# B&R Automation Studio project NewPendant_NG4_11_05_25A (part 7)

```c
				// Dodane - Nie ma Xcmd Stop w TRVL_BPV_POS
				if((TVL_ROT_Param_Set[0].Mode == 2) // with only position
					|| (TVL_ROT_Param_Set[0].Mode == 3)) // with interrupt
					Process[m->pCfg->HeadCfg.TVL.PROC_Indx].xCMD = 0;
			}
			*/

///////////////////////////////////////////////////////////////////////////
/// Nowosc Index wczesniej

			if((curCalib->GenSetup[SETUP_EXTRAS]&0x4)){

				switch(curCalib->GenSetup[SETUP_HEAD_SETUP] ){

						default:

							if(curCalib->GenSetup[SETUP_INDX_ENBL] == 3){ // In OSc

								if(INDEX_Param_Set[0].pStepDist){

									Process[m->pCfg->HeadCfg.OSC.PROC_Indx].xCMD = prcsSTEPneg; // Quick Step with delay

									if(curCalib->GenSetup[SETUP_INDX_DIR])
										Process[m->pCfg->HeadCfg.OSC.PROC_Indx].fParam[1] = (*INDEX_Param_Set[0].pStepDist);
									else
										Process[m->pCfg->HeadCfg.OSC.PROC_Indx].fParam[1] = (*INDEX_Param_Set[0].pStepDist) * (-1.0);

									KK_Catched = 133;

									//m->SeqStep++;
								}
								//else
									//m->SeqStep = 203;

							}

							else if(curCalib->GenSetup[SETUP_INDX_ENBL] == 1){

								if(INDEX_Param_Set[0].pStepDist){
									Process[m->pCfg->HeadCfg.INDX.PROC_Indx].xCMD = prcsSTEPpos;

									if(curCalib->GenSetup[SETUP_INDX_DIR])
										Process[m->pCfg->HeadCfg.INDX.PROC_Indx].fParam[1] = (*INDEX_Param_Set[0].pStepDist);
									else
										Process[m->pCfg->HeadCfg.INDX.PROC_Indx].fParam[1] = (*INDEX_Param_Set[0].pStepDist) * (-1.0);

									m->SeqStep++;

								}
								//else
									//m->SeqStep = 203;

							}
							//else
								//m->SeqStep = 203;

						break;

					}

			}

/////////////////////////////////////////////////////////////////////////
#ifdef EXTENDED_LOGS

			LogTxt(&LogMgr, "Path %d Done: %.2f" , (UDINT)File_RW._int.PathDoneCnt, ABS_TVL_Pos);
#else
			LogTxt(&LogMgr, "Path %d Done" , (UDINT)File_RW._int.PathDoneCnt);

#endif

			//TimerStart(&WF_Catch_TMR, curCfg->Param[parWF_RampDwn].val[0]);
			m->SeqStep++;

		break;

		case 201:

			// Always Coolant On
			if (!m->TestMode)
			{
				if (Process[m->pCfg->HeadCfg.COOL.PROC_Indx].Status != prcsSTATUS_Run)
					Process[m->pCfg->HeadCfg.COOL.PROC_Indx].xCMD = prcsSTART;
			}

			ret = 5; // Preparing To Stop

			if (StopBtn)
			{
#ifdef EXTENDED_LOGS

				LogTxt(&LogMgr, "Quick stop %.2f" , ABS_TVL_Pos);
#else
				LogTxt(&LogMgr, "Quick stop");
#endif
				m->SeqStep = 254;			// Quick Stop
			}

			status = 1;

			if (Process[m->pCfg->HeadCfg.TVL.PROC_Indx].Status != prcsSTATUS_Stopped){ // stopped by end of travel
				status = 0;
			}
			if (Process[m->pCfg->HeadCfg.OSC.PROC_Indx].Status != prcsSTATUS_Stopped)
				status = 0;

			if (Process[m->pCfg->HeadCfg.AVC.PROC_Indx].Status != prcsSTATUS_Stopped)
				status = 0;

			if (Process[m->pCfg->HeadCfg.WF.PROC_Indx].Status != prcsSTATUS_Stopped)
				status = 0;

			//if (Process[m->pCfg->HeadCfg.GAS.PROC_Indx].Status != prcsSTATUS_Stopped)
				//status = 0;

			if (Process[m->pCfg->HeadCfg.WP.PROC_Indx].Status != prcsSTATUS_Stopped)
				status = 0;

			if (Process[m->pCfg->HeadCfg.TIG.PROC_Indx].Status != prcsSTATUS_Stopped)
				status = 0;

			if (Process[m->pCfg->HeadCfg.HW.PROC_Indx].Status != prcsSTATUS_Stopped)
				status = 0;

			if (status)
			{

#ifdef EXTENDED_LOGS

				LogTxt(&LogMgr, "M:All%d Stop: %.2f" ,(UDINT) m->ToolHeadID, ABS_TVL_Pos);

#endif

				if(!(curCalib->GenSetup[SETUP_EXTRAS]&0x4)){

					switch(curCalib->GenSetup[SETUP_HEAD_SETUP] ){

						/*
						case BPV_v2_MPGH:
						case BPV_v2_MPGV:

						case BPV_v2_MPBO:

							if(curCalib->GenSetup[SETUP_INDX_ENBL] == 3){ // In OSc

								if(INDEX_Param_Set[0].pStepDist){

									Process[m->pCfg->HeadCfg.OSC.PROC_Indx].xCMD = prcsSTEPpos;

									if(curCalib->GenSetup[SETUP_INDX_DIR])
										Process[m->pCfg->HeadCfg.OSC.PROC_Indx].fParam[1] = (*INDEX_Param_Set[0].pStepDist);
									else
										Process[m->pCfg->HeadCfg.OSC.PROC_Indx].fParam[1] = (*INDEX_Param_Set[0].pStepDist) * (-1.0);

									KK_Catched = 133;

									m->SeqStep++;
								}
								else
									m->SeqStep = 203;

							}
							else
								m->SeqStep = 203;

						break;
						*/

						default:

							if(curCalib->GenSetup[SETUP_INDX_ENBL] == 3){ // In OSc

								if(INDEX_Param_Set[0].pStepDist){

									Process[m->pCfg->HeadCfg.OSC.PROC_Indx].xCMD = prcsSTEPpos;

									if(curCalib->GenSetup[SETUP_INDX_DIR])
										Process[m->pCfg->HeadCfg.OSC.PROC_Indx].fParam[1] = (*INDEX_Param_Set[0].pStepDist);
									else
										Process[m->pCfg->HeadCfg.OSC.PROC_Indx].fParam[1] = (*INDEX_Param_Set[0].pStepDist) * (-1.0);

									KK_Catched = 133;

									m->SeqStep++;
								}
								else
									m->SeqStep = 203;

							}

							else if(curCalib->GenSetup[SETUP_INDX_ENBL] == 1){

								if(INDEX_Param_Set[0].pStepDist){
									Process[m->pCfg->HeadCfg.INDX.PROC_Indx].xCMD = prcsSTEPpos;

									if(curCalib->GenSetup[SETUP_INDX_DIR])
										Process[m->pCfg->HeadCfg.INDX.PROC_Indx].fParam[1] = (*INDEX_Param_Set[0].pStepDist);
									else
										Process[m->pCfg->HeadCfg.INDX.PROC_Indx].fParam[1] = (*INDEX_Param_Set[0].pStepDist) * (-1.0);

									m->SeqStep++;

								}
								else
									m->SeqStep = 203;

							}
							else
								m->SeqStep = 203;

						break;

					}

					}

			}

		break;

		case 202:

			// Always Coolant On
			if (!m->TestMode)
			{
				if (Process[m->pCfg->HeadCfg.COOL.PROC_Indx].Status != prcsSTATUS_Run)
					Process[m->pCfg->HeadCfg.COOL.PROC_Indx].xCMD = prcsSTART;
			}

			if (StopBtn)
			{
				LogTxt(&LogMgr, "Quick stop");

				m->SeqStep			= 254;			// Quick Stop
				break;
			}

			if(Process[m->pCfg->HeadCfg.INDX.PROC_Indx].Status == prcsSTATUS_Stopped
				&& Process[m->pCfg->HeadCfg.OSC.PROC_Indx].Status == prcsSTATUS_Stopped){

				TimerStart(&m->sm.Tmr1, 0.1);
				m->SeqStep++;

			}

		break;

		case 203:
			// Always Coolant On
			if (StopBtn)
			{
				LogTxt(&LogMgr, "Halt stop");

				m->SeqStep			= 254;			// Quick Stop
				break;
			}

			if (!m->TestMode)
			{
				if (Process[m->pCfg->HeadCfg.COOL.PROC_Indx].Status != prcsSTATUS_Run)
					Process[m->pCfg->HeadCfg.COOL.PROC_Indx].xCMD = prcsSTART;
			}

			if(Process[m->pCfg->HeadCfg.TVL.PROC_Indx].Status == prcsSTATUS_Stopped){

				LogTxt(&LogMgr, "M: Cyc. Time %.2f" , GlobalTimer);
				m->SeqStep++;
			}

		break;

		case 204:

			// Always Coolant On
			if (!m->TestMode)
			{
				if (Process[m->pCfg->HeadCfg.COOL.PROC_Indx].Status != prcsSTATUS_Run)
					Process[m->pCfg->HeadCfg.COOL.PROC_Indx].xCMD = prcsSTART;
			}

			ret = 5; // Preparing To Stop

			if (StopBtn)
			{
				LogTxt(&LogMgr, "Quick stop");
				m->SeqStep = 254;			// Quick Stop
				//m->SeqStep = 205;			// Normal Stop
				break;
			}

			// Check if Index move done
			if (1)
			{

				if((abs(m->curSegm[ACT_TVL_DIST] - Process[m->pCfg->HeadCfg.TVL.PROC_Indx].Param[3]) < 10)
				//if((Process[m->pCfg->HeadCfg.TVL.PROC_Indx].Status == prcsSTATUS_Stopped)
					&& (m->SubSeqStep == 2)) // IMPORTANT - head swap is only when was rewrap before
				{

					m->SubSeqStep = 1;

					if (curCfg->Param_ENUM[parENUM_PathMode].val[0] == 0.0)
						m->ToolHeadID = !m->ToolHeadID;

					if (curCfg->Param_ENUM[parENUM_TVL_MODE].val[0] == 0)
					{ // Relative Move
						if (TVL_ROT_Param_Set[0].pEncoder)
							OLD_MTR_POS[TVL_ENC_HOME] = *TVL_ROT_Param_Set[0].pEncoder;
					}
					AutoStartEnable = 1;
					m->SeqStep++;

				}

				else
				{
					m->SeqStep = 254;
				}

			}

		break;

		case 205:

			if(curCfg->Param[parGEN_WeldProgramRepeat].val[0] > 0)
				File_RW._int.PathDoneCnt++;
			else
				File_RW._int.PathDoneCnt = 0;

			newFile = 0;

			if (curCfg->Param_ENUM[parENUM_WeldProgramLinkMode].val[0] > 0.0)
			{

				if (curCfg->Param[parGEN_WeldProgramRepeat].val[0] == 0.0)
				{

					if (strlen(curCfg->NextProgramName) > 0)
					{

						if (!strstr(curCfg->NextProgramName, "NONE"))
						{ // Not None
							TakeNextWeldProgram(hmi);
							newFile 			= 1;

						}

					}

				}

				else
				{

					if (File_RW._int.PathDoneCnt > (UINT)curCfg->Param[parGEN_WeldProgramRepeat].val[0] )
					{

						if (strlen(curCfg->NextProgramName) > 0)
						{

							if (!strstr(curCfg->NextProgramName, "NONE"))
							{ // Not None
								TakeNextWeldProgram(hmi);
								newFile 			= 1;
							}

						}

					}

				}

			}

			if (newFile)
				m->SeqStep = 206;
			else
				m->SeqStep = 207;

		break;

		case 206:
			if (File_RW.CMD == 0)
			{

				if (File_RW.Error)
					m->SeqStep = 206;

				else
				{
					AutoStartEnable = 1;
					m->SeqStep = 207;

				}
			}

		break;

		case 207:

			AutoStartEnable = 1;

			if (File_RW._int.PathDoneCnt > (UINT)curCfg->Param[parGEN_WeldProgramRepeat].val[0] )
			{
				File_RW._int.PathDoneCnt = (UINT)curCfg->Param[parGEN_WeldProgramRepeat].val[0];

				AutoStartEnable 	= 0;
			}

			m->SeqStep++;

		break;

		case 208:
			///////////////////////////////////
			//Auto Start
			if (curCalib->GenSetup[SETUP_AUTO_START] && AutoStartEnable)
			{
				TimerStart(&m->sm.Tmr1, curCalib->GenFloatValue[SETUP_FLOAT_AUTOSTART_DLY]);
				m->SeqStep = 220;

			}
			else
				m->SeqStep = 254;

		break;

		case 210:

			if (StopBtn)
			{
				LogTxt(&LogMgr, "Quick stop");

				m->SeqStep = 254;			// Quick Stop

			}
			else if (Process[m->pCfg->HeadCfg.TVL.PROC_Indx].Status == prcsSTATUS_Stopped) // stopped by end of travel
				m->SeqStep = 0;

		break;

		case 220:

			if (StopBtn)
			{
				LogTxt(&LogMgr, "Quick stop");

				m->SeqStep = 254;			// Quick Stop
				break;
			}
			else if(!TimerIsTimeOut(&m->sm.Tmr1))
				break;

			GlobalTimer = 0;

			//WF_TVL_Diff = 0;
			LogTxt(&LogMgr, "Auto Repeat");
			AutoStartBtn = 1;
			m->SeqStep = 0;

		break;

		case 254:

			for (i = 0; i < PROCESS_NUM; i++)
			{ // beside PROC_COOL
				if (i != PROC_COOL)
					Process[i].xCMD = prcsHalt;
			}

			Process[m->pCfg->HeadCfg.OSC.PROC_Indx].Param[0] = 1; // STop without ramp
			Process[m->pCfg->HeadCfg.OSC.PROC_Indx].xCMD = prcsQuickSTOP; // return to center position
			Process[m->pCfg->HeadCfg.GAS.PROC_Indx].xCMD = prcsSTOP; // maintain gas
			m->SeqStep++;

		break;

		default:

			if(curCfg->Param_ENUM[parENUM_AVC_Mode].val[0] != 3) // AVC Mode NOT LOCKED !
				Process[m->pCfg->HeadCfg.AVC.PROC_Indx].Param[0] = 0;

			if (StopBtn)
			{
				LogTxt(&LogMgr, "Halt stop");

				for (i = 0; i < PROCESS_NUM; i++)
				{ // beside PROC_COOL
					if (i!= PROC_COOL && i!= PROC_OSC)
						Process[i].xCMD = prcsHalt;
				}

				Process[m->pCfg->HeadCfg.GAS.PROC_Indx].xCMD = prcsSTOP; // maintain gas
				m->SeqStep			= 0;

			}

			if (Process[m->pCfg->HeadCfg.OSC.PROC_Indx].Status == prcsSTATUS_Stopped)
				m->SeqStep = 0;

			if (m->SeqStep == 0)
			{
				// Load new AVC param from new file
				TML_MTR_INST[m->pCfg->HeadCfg.AVC.TML_A_Indx]._cfg.signFilter =	curCfg->Param[parAVC_FbkFilter].val[0];
			}

		break;

		}

		//if((Process[m->pCfg->HeadCfg.TVL.PROC_Indx].Status == prcsSTATUS_Stopped))
		//StopBtn_Latch = 0;
		////////////////////////////
		TimerExecute(&WireDisable_TMR);
		TimerExecute(&WF_Catch_TMR);

		return ret;
	}

		/*********************************************************/
			/****	Process parameters assigments	************************/

	DINT MasterSequence_Contin_OneWay_dobra_alebezWeldIndex(MASTER_typ * m, HMI_typ * hmi, plcbit StartBtn, plcbit StopBtn)
	{
	int 			i;
	char			status;
	DINT			ret;
	DINT			d;
	USINT			newFile;

	//Cfg_typ *cfg;
	CurCfg_typ *	curCfg;

	//CurCalib_typ *curCalib , *defCalib;
	//Scaled_Var_obj *var;
	//cfg = (Cfg_typ*) m->pCfg;
	curCfg				= (CurCfg_typ *)
	m->pCurCfg;

	//curCalib = (CurCalib_typ*) m->pCalib;
	//defCalib = (CurCalib_typ*) m->pDefaultCalib;
	//var = (Scaled_Var_obj*) m->pScaledVar;
	m->TestMode 		= intrf->TestMode;

	ret 				= 0;

	if((hmi->curHeadID == 0xFFFE)){ // Screen RUn or Alter Run

		if(intrf->GlblBtnCmd[0] &ANDR_BTN_UP){

			AVC_Param_Set[0].BoostCmd = 1;
			PS_Param_Set[0].BoostCmd = 1;
			TVL_ROT_Param_Set[0].BoostCmd = 1;
			WIRE_Param_Set[0].BoostCmd = 1;
			WIRE_Param_Set[1].BoostCmd = 1;

		}
		else if(intrf->GlblBtnCmd[0] &ANDR_BTN_DOWN){

			AVC_Param_Set[0].BoostCmd = 2;
			PS_Param_Set[0].BoostCmd = 2;
			TVL_ROT_Param_Set[0].BoostCmd = 2;
			WIRE_Param_Set[0].BoostCmd = 2;
			WIRE_Param_Set[1].BoostCmd = 2;

		}
		else{

			AVC_Param_Set[0].BoostCmd = 0;
			PS_Param_Set[0].BoostCmd = 0;
			TVL_ROT_Param_Set[0].BoostCmd = 0;
			WIRE_Param_Set[0].BoostCmd = 0;
			WIRE_Param_Set[1].BoostCmd = 0;

		}
	}
	else{

		AVC_Param_Set[0].BoostCmd = 0;
		PS_Param_Set[0].BoostCmd = 0;
		TVL_ROT_Param_Set[0].BoostCmd = 0;
		WIRE_Param_Set[0].BoostCmd = 0;
		WIRE_Param_Set[1].BoostCmd = 0;

	}

	/////////
	/////////
	//(!intrf->_intr._GlblBtnCmd[0] && (intrf->GlblBtnCmd[0] &ANDR_BTN_STOP)
	/*
	if (StopBtn)
	{
		AutoStartBtn		= 0;

		if (TimerIsTimeOut(&DoubleStop_TMR))
			TimerStart(&DoubleStop_TMR, 0.5);
		else
			DoubleStopBtn_Latch = 1;
	}

	if (StopBtn)
		StopBtn_Latch = 1;

	*/

	if (Process[m->pCfg->HeadCfg.TVL.PROC_Indx].Status != prcsSTATUS_Stopped)
	{
		if(m->SubSeqStep == 1 )// Weld to Target
		{
			if(abs(m->curSegm[ACT_TVL_DIST] - Process[m->pCfg->HeadCfg.TVL.PROC_Indx].Param[0]) < 10)
				m->SubSeqStep = 2;
		}
	}

	if ((Process[m->pCfg->HeadCfg.TVL.PROC_Indx].Status == prcsSTATUS_Stopped) ||
	(Process[m->pCfg->HeadCfg.TVL.PROC_Indx].Status == prcsSTATUS_ReturnDly)){

		if(DoubleStopBtn_Latch){
			if(m->SubSeqStep > 0){
				AutoStartBtn = 0;
				m->SubSeqStep = 0;
			}
			else
				m->SubSeqStep = 1;

		}
	}
	DoubleStopBtn_Latch = 0;

	if(curCfg->Param_ENUM[parENUM_TVL_MODE].val[0] == 3) // Continues welding
		m->SubSeqStep = 0;

	if (StopBtn_Latch)
		Process[m->pCfg->HeadCfg.TVL.PROC_Indx].Param[2] = 0; // No Auto Stop and Not Rewrap

	//////////////////////////
	////////////////////////////
	if (m->SeqStep > 0)
		GlobalTimer += 0.0512; // Timer based on task class

	//////////////

		//	 MASTER SEQUENCE  //
	switch (m->SeqStep)
	{
		case 0:

			Cont_Stop_By_End = 0;
			//////////////////////////////////////
			if(curCfg->Param[parGEN_WeldProgramRepeat].val[0] == 0.0)
				File_RW._int.PathDoneCnt = 0;

			// Reset Disable when was in Test Mode
			Process[m->pCfg->HeadCfg.AVC.PROC_Indx].Disable &= 0xFD;
			Process[m->pCfg->HeadCfg.OSC.PROC_Indx].Disable &= 0xFD;
			Process[m->pCfg->HeadCfg.TVL.PROC_Indx].Disable &= 0xFD;
			Process[m->pCfg->HeadCfg.TIG.PROC_Indx].Disable &= 0xFD;
			Process[m->pCfg->HeadCfg.HW.PROC_Indx].Disable &= 0xFD;
			StopBtn_Latch = 0;

			// AVC Locked is OFF

			//if(curCfg->Param_ENUM[parENUM_AVC_Mode].val[0] != 3) // AVC Mode NOT LOCKED !
				//Process[m->pCfg->HeadCfg.AVC.PROC_Indx].Param[0] = 0;

			if(StartBtn && !Check_OSC_Amplt_and_Center())
				break;

			if (StopBtn)
			{
				LogTxt(&LogMgr, "Quick stop");
				m->SeqStep = 254;			// Halt Stop
				break;
			}

			status = 1;

			if (//(Process[m->pCfg->HeadCfg.GAS.PROC_Indx].Status != prcsSTATUS_Stopped)
				(Process[m->pCfg->HeadCfg.AVC.PROC_Indx].Status != prcsSTATUS_Stopped) ||
				(Process[m->pCfg->HeadCfg.OSC.PROC_Indx].Status != prcsSTATUS_Stopped) ||
				(Process[m->pCfg->HeadCfg.TVL.PROC_Indx].Status != prcsSTATUS_Stopped) ||
				(Process[m->pCfg->HeadCfg.WF.PROC_Indx].Status != prcsSTATUS_Stopped) ||
				(Process[m->pCfg->HeadCfg.WP.PROC_Indx].Status != prcsSTATUS_Stopped))
				status = 0;

			if (status)
			{

				if (!ErrorMgr.Error)
				{
					ret = 1;		// Raedy To Run

					if((intrf->GlblBtnCmd[0] &ANDR_BTN_HOME) && StartBtn){

						Process[m->pCfg->HeadCfg.TVL.PROC_Indx].Param[3] = 0;
						Process[m->pCfg->HeadCfg.TVL.PROC_Indx].Param[2] = 2; //only rewrap
						Process[m->pCfg->HeadCfg.TVL.PROC_Indx].xCMD = prcsSTART;
						m->SeqStep = 210;

					}

					//if ((StartBtn || AutoStartBtn) && (XMLHelper.xCmd != XML_CMD_READ))
					//if (StartBtn || AutoStartBtn)
					else if ((StartBtn || AutoStartBtn) && ((Weld_Report_Status < 2) || ((curCalib->GenSetup[SETUP_EXTRAS]&0x1) == 0)))
					{
						Weld_Report_Status = 1;
						AutoStartBtn = 0;

						if (m->SubSeqStep == 2)
						{ // Rewrap

							if (curCalib->GenSetup[SETUP_SOUND_DELAY] || curCalib->GenSetup[SETUP_AUTO_START])
								TimerStart(&m->sm.Tmr1, curCalib->GenFloatValue[SETUP_FLOAT_SOUND_TM]);

							else
								TimerStart(&m->sm.Tmr1, 0.1);

							m->SeqStep = 150;

						}
						else
						{

						GlobalTimer 		= 0;

						LogTxt(&LogMgr, "PreProcess start");

						if (curCalib->GenSetup[SETUP_SOUND_DELAY] || curCalib->GenSetup[SETUP_AUTO_START])
							TimerStart(&m->sm.Tmr1, curCalib->GenFloatValue[SETUP_FLOAT_SOUND_TM]);
						else
							TimerStart(&m->sm.Tmr1, 0.1);

							m->SeqStep++;

						}
					}

					/*
					else if ((StartBtn || AutoStartBtn) && (XMLHelper.xCmd == XML_CMD_READ)){

						strcpy(hmi->pMessage[0], " FILE OPER. \n ");
						strcpy(hmi->pMessage[1], File_RW.fileName);
						strcpy(hmi->pMessage[2], "Is Loading");
						strcpy(hmi->pMessage[3] ,"Wait for finish");

						Set_Message(hmi , 0.1);

					}
					*/
				}

			}
			else
			{
				if (StopBtn)
				{
					LogTxt(&LogMgr, "Some Prcs aborted");
					m->SeqStep = 254;
				}

			}

		break;

		case 1:
		// Always Coolant On

			Cont_Stop_By_End = 0;

			if (!m->TestMode)
			{
				if (Process[m->pCfg->HeadCfg.COOL.PROC_Indx].Status != prcsSTATUS_Run)
					Process[m->pCfg->HeadCfg.COOL.PROC_Indx].xCMD = prcsSTART;
			}

			ret = 2; // Preparig To Run

			if (StopBtn)
			{
				LogTxt(&LogMgr, "Some Prcs aborted");
				m->SeqStep = 254;
			}
			else if (ErrorMgr.Error)
				m->SeqStep = 100;

			else if (!TimerIsTimeOut(&m->sm.Tmr1))
				break;

			else
			{
				if (!m->TestMode)
				{
					Process[m->pCfg->HeadCfg.GAS.PROC_Indx].xCMD = prcsSTART;
					Process[m->pCfg->HeadCfg.COOL.PROC_Indx].xCMD = prcsSTART;
				}

				if (m->TestMode)
				{

					//Process[m->pCfg->HeadCfg.AVC.PROC_Indx].Disable |= 0x02 ;
					Process[m->pCfg->HeadCfg.AVC.PROC_Indx].TestMode = 1;
					Process[m->pCfg->HeadCfg.TIG.PROC_Indx].Disable |= 0x02;
					Process[m->pCfg->HeadCfg.HW.PROC_Indx].Disable |= 0x02;

				}
				else
				{

					if ((Process[m->pCfg->HeadCfg.GAS.PROC_Indx].Status == prcsSTATUS_Run) &&
					(Process[m->pCfg->HeadCfg.COOL.PROC_Indx].Status == prcsSTATUS_Run))
					{
						//Process[m->pCfg->HeadCfg.AVC.PROC_Indx].Disable &= 0xFD ;
						Process[m->pCfg->HeadCfg.AVC.PROC_Indx].TestMode = 0;
						Process[m->pCfg->HeadCfg.TIG.PROC_Indx].Disable &= 0xFD;
						Process[m->pCfg->HeadCfg.HW.PROC_Indx].Disable &= 0xFD;

					}
					else
						break;

				}

				Process[m->pCfg->HeadCfg.AVC.PROC_Indx].xCMD = prcsSTART;

				//if(!m->TestMode)
				Process[m->pCfg->HeadCfg.TIG.PROC_Indx].xCMD = prcsForceON;

				LogTxt(&LogMgr, "ARC start");

				m->SeqStep++;

			}

		break;

		case 2:

			// Always Coolant On
			if (!m->TestMode)
			{
				if (Process[m->pCfg->HeadCfg.COOL.PROC_Indx].Status != prcsSTATUS_Run)
					Process[m->pCfg->HeadCfg.COOL.PROC_Indx].xCMD = prcsSTART;
			}

			ret = 2; // Preparig To Run

			if (StopBtn)
			{
				LogTxt(&LogMgr, "Some Prcs aborted");
				m->SeqStep			= 254;
			}

			///////////////////////////
			else if (ErrorMgr.Error)
				m->SeqStep = 100;

			else if ((Process[m->pCfg->HeadCfg.AVC.PROC_Indx].Status == prcsSTATUS_Run)
					|| (Process[m->pCfg->HeadCfg.AVC.PROC_Indx].Status == prcsSTATUS_AVC_OK))
			{

				Process[m->pCfg->HeadCfg.OSC.PROC_Indx].xCMD = prcsSTART;
				Process[m->pCfg->HeadCfg.OSC.PROC_Indx].Param[0] = 0; // Start with ramp
				Process[m->pCfg->HeadCfg.TIG.PROC_Indx].xCMD = prcsSTART;

				/*	TVL */
				Process[m->pCfg->HeadCfg.TVL.PROC_Indx].Param[2] = m->SubSeqStep;
				Process[m->pCfg->HeadCfg.TVL.PROC_Indx].xCMD = prcsSTART;

#ifdef EXTENDED_LOGS
				LogTxt(&LogMgr, "M:TVL%d Start: %.2f" , (UDINT) m->ToolHeadID , ABS_TVL_Pos);
#endif
				StartPos = 0;

				CalculateRunOverlap_Cont_OneWay();

				if (!m->WireDisabled)
				{
					// if prcsStart then Param[0] = 0 is set in Wire process - jus in case
					//Process[m->pCfg->HeadCfg.WF.PROC_Indx].Param[0] = 0; // start with full ramp
					Process[m->pCfg->HeadCfg.WF.PROC_Indx].xCMD = prcsSTART;
					//Process[m->pCfg->HeadCfg.WP.PROC_Indx].Param[0] = 0; // start with full ramp
					Process[m->pCfg->HeadCfg.WP.PROC_Indx].xCMD = prcsSTART;
					Process[m->pCfg->HeadCfg.HW.PROC_Indx].xCMD = prcsSTART;
				}

				LogTxt(&LogMgr, "ARC established");

				TimerStart(&WireDisable_TMR, 3.0);

				m->SeqStep++;

			}

		break;

		case 3:
			// Always Coolant On
			if (!m->TestMode)
			{
				if (Process[m->pCfg->HeadCfg.COOL.PROC_Indx].Status != prcsSTATUS_Run)
					Process[m->pCfg->HeadCfg.COOL.PROC_Indx].xCMD = prcsSTART;
			}

			WireDisableInable(WireDisable_TMR.Q);
			Process[m->pCfg->HeadCfg.TIG.PROC_Indx].Param[0] = Process[m->pCfg->HeadCfg.OSC.PROC_Indx].subStatus;
			Process[m->pCfg->HeadCfg.HW.PROC_Indx].Param[0] = Process[m->pCfg->HeadCfg.OSC.PROC_Indx].subStatus;
			ret = 3; //  Run

			//if (actRot != _actRot)
				//TakeNextWeldProgram(hmi);

			_actRot = actRot;

			if (Process[m->pCfg->HeadCfg.TVL.PROC_Indx].subStatus == 1)
			{ // End of travel reached
				//LogTxt(&LogMgr, "Path Done");
				//LogTxt(&LogMgr, "Path Done: %.2f" , ABS_TVL_Pos);

				Weld_Report_Status = 2;

				m->SeqStep = 200;

			}

			if (StopBtn)
			{
				/*
				LogTxt(&LogMgr, "Process stop");
				//Process[m->pCfg->HeadCfg.TVL.PROC_Indx].xCMD = prcsSTOP;
				m->SeqStep = 200;
				*/
				if(Cont_Stop_By_End){
					LogTxt(&LogMgr, "Process stop by Operator");
					Cont_Stop_By_End = 0;
					m->SeqStep = 200;
				}
				else
					Cont_Stop_By_End = 1;

			}
			else if (ErrorMgr.Error || m->ESTOP)
			{
				LogTxt(&LogMgr, "Process Error");
				m->SeqStep = 100;
			}

		break;

		case 100:
			// Always Coolant On
			if (!m->TestMode)
			{
				if (Process[m->pCfg->HeadCfg.COOL.PROC_Indx].Status != prcsSTATUS_Run)
					Process[m->pCfg->HeadCfg.COOL.PROC_Indx].xCMD = prcsSTART;
			}

			Process[m->pCfg->HeadCfg.TVL.PROC_Indx].xCMD = prcsHalt;
			Process[m->pCfg->HeadCfg.OSC.PROC_Indx].xCMD = prcsHalt;
			Process[m->pCfg->HeadCfg.AVC.PROC_Indx].xCMD = prcsHalt;
			Process[m->pCfg->HeadCfg.WF.PROC_Indx].xCMD = prcsHalt;
			Process[m->pCfg->HeadCfg.WP.PROC_Indx].xCMD = prcsHalt;
			Process[m->pCfg->HeadCfg.TIG.PROC_Indx].xCMD = prcsHalt;
			Process[m->pCfg->HeadCfg.HW.PROC_Indx].xCMD = prcsHalt;
			Process[m->pCfg->HeadCfg.GAS.PROC_Indx].xCMD = prcsSTOP;

			//Process[m->pCfg->HeadCfg.COOL.PROC_Indx].xCMD = prcsHalt;
			switch (ErrorMgr.Error)
			{
				case ERROR_FATAL:
					m->SeqStep++;
				break;

				case ERROR_MOTOR:
					m->SeqStep++;
				break;

				case ERROR_MOTOR_INIT:
					m->SeqStep++;
				break;

				case ERROR_TIG_PROC:
					m->SeqStep++;
				break;

				default:
					m->SeqStep++;
				break;
			}

		break;

		case 101:
			ret = 4; // Preparig To Stop in Halt Mode

			if (StopBtn)
			{
				for (i = 0; i < PROCESS_NUM; i++)
				{
					if (i != PROC_COOL)
						Process[i].xCMD = prcsHalt;
				}
				Process[m->pCfg->HeadCfg.GAS.PROC_Indx].xCMD = prcsSTOP; // maintain gas
			}

			status = 1;

			if (Process[m->pCfg->HeadCfg.TVL.PROC_Indx].Status != prcsSTATUS_Stopped)
				status = 0;

			if (Process[m->pCfg->HeadCfg.OSC.PROC_Indx].Status != prcsSTATUS_Stopped)
				status = 0;

			if (Process[m->pCfg->HeadCfg.AVC.PROC_Indx].Status != prcsSTATUS_Stopped)
				status = 0;

			if (Process[m->pCfg->HeadCfg.WF.PROC_Indx].Status != prcsSTATUS_Stopped)
				status = 0;

			if (Process[m->pCfg->HeadCfg.GAS.PROC_Indx].Status != prcsSTATUS_Stopped)
				status = 0;

			if (Process[m->pCfg->HeadCfg.WP.PROC_Indx].Status != prcsSTATUS_Stopped)
				status = 0;

			if (Process[m->pCfg->HeadCfg.TIG.PROC_Indx].Status != prcsSTATUS_Stopped)
				status = 0;

			if (Process[m->pCfg->HeadCfg.HW.PROC_Indx].Status != prcsSTATUS_Stopped)
				status = 0;

			if (status)
			{
				LogTxt(&LogMgr, "Prc Final stopped");
				m->SeqStep = 254;
			}

		break;

		case 150:

			if (StopBtn)
			{
				LogTxt(&LogMgr, "Quick stop");
				m->SeqStep = 254;			// Quick Stop
				break;
			}

			if (!TimerIsTimeOut(&m->sm.Tmr1))
				break;

			/*	TVL */
			Process[m->pCfg->HeadCfg.TVL.PROC_Indx].Param[2] = m->SubSeqStep;
			Process[m->pCfg->HeadCfg.TVL.PROC_Indx].xCMD = prcsSTART;
			StartPos = 0;

			CalculateRunOverlap_Cont_OneWay();

			m->SeqStep = 202;

		break;

		case 200:

			// Always Coolant On
			if (!m->TestMode)
			{
				if (Process[m->pCfg->HeadCfg.COOL.PROC_Indx].Status != prcsSTATUS_Run)
					Process[m->pCfg->HeadCfg.COOL.PROC_Indx].xCMD = prcsSTART;
			}

			for (i = 0; i < PROCESS_NUM; i++)
			{
				if ((i != PROC_COOL)) //&&( i != m->pCfg->HeadCfg.TVL.PROC_Indx))
					Process[i].xCMD = prcsSTOP;

			}
#ifdef EXTENDED_LOGS

			LogTxt(&LogMgr, "Path %d Done: %.2f" , (UDINT)File_RW._int.PathDoneCnt, ABS_TVL_Pos);
#else
			LogTxt(&LogMgr, "Path %d Done" , (UDINT)File_RW._int.PathDoneCnt);

#endif

			//TimerStart(&WF_Catch_TMR, curCfg->Param[parWF_RampDwn].val[0]);
			m->SeqStep++;

		break;

		case 201:

			// Always Coolant On
			if (!m->TestMode)
			{
				if (Process[m->pCfg->HeadCfg.COOL.PROC_Indx].Status != prcsSTATUS_Run)
					Process[m->pCfg->HeadCfg.COOL.PROC_Indx].xCMD = prcsSTART;
			}

			ret = 5; // Preparing To Stop

			if (StopBtn)
			{
#ifdef EXTENDED_LOGS

				LogTxt(&LogMgr, "Quick stop %.2f" , ABS_TVL_Pos);
#else
				LogTxt(&LogMgr, "Quick stop");
#endif
				m->SeqStep = 254;			// Quick Stop
			}

			status = 1;

			if (Process[m->pCfg->HeadCfg.TVL.PROC_Indx].Status != prcsSTATUS_Stopped){ // stopped by end of travel
				status = 0;
			}
			if (Process[m->pCfg->HeadCfg.OSC.PROC_Indx].Status != prcsSTATUS_Stopped)
				status = 0;

			if (Process[m->pCfg->HeadCfg.AVC.PROC_Indx].Status != prcsSTATUS_Stopped)
				status = 0;

			if (Process[m->pCfg->HeadCfg.WF.PROC_Indx].Status != prcsSTATUS_Stopped)
				status = 0;

			//if (Process[m->pCfg->HeadCfg.GAS.PROC_Indx].Status != prcsSTATUS_Stopped)
				//status = 0;

			if (Process[m->pCfg->HeadCfg.WP.PROC_Indx].Status != prcsSTATUS_Stopped)
				status = 0;

			if (Process[m->pCfg->HeadCfg.TIG.PROC_Indx].Status != prcsSTATUS_Stopped)
				status = 0;

			if (Process[m->pCfg->HeadCfg.HW.PROC_Indx].Status != prcsSTATUS_Stopped)
				status = 0;

			if (status)
			{

#ifdef EXTENDED_LOGS

				LogTxt(&LogMgr, "M:All%d Stop: %.2f" ,(UDINT) m->ToolHeadID, ABS_TVL_Pos);

#endif
				switch(curCalib->GenSetup[SETUP_HEAD_SETUP] ){

					/*
					case BPV_v2_MPGH:
					case BPV_v2_MPGV:

					case BPV_v2_MPBO:

						if(curCalib->GenSetup[SETUP_INDX_ENBL] == 3){ // In OSc

							if(INDEX_Param_Set[0].pStepDist){

								Process[m->pCfg->HeadCfg.OSC.PROC_Indx].xCMD = prcsSTEPpos;

								if(curCalib->GenSetup[SETUP_INDX_DIR])
									Process[m->pCfg->HeadCfg.OSC.PROC_Indx].fParam[1] = (*INDEX_Param_Set[0].pStepDist);
								else
									Process[m->pCfg->HeadCfg.OSC.PROC_Indx].fParam[1] = (*INDEX_Param_Set[0].pStepDist) * (-1.0);

								KK_Catched = 133;

								m->SeqStep++;
							}
							else
								m->SeqStep = 203;

						}
						else
							m->SeqStep = 203;

					break;
					*/

					default:

						if(curCalib->GenSetup[SETUP_INDX_ENBL] == 3){ // In OSc

							if(INDEX_Param_Set[0].pStepDist){

								Process[m->pCfg->HeadCfg.OSC.PROC_Indx].xCMD = prcsSTEPpos;

								if(curCalib->GenSetup[SETUP_INDX_DIR])
									Process[m->pCfg->HeadCfg.OSC.PROC_Indx].fParam[1] = (*INDEX_Param_Set[0].pStepDist);
								else
									Process[m->pCfg->HeadCfg.OSC.PROC_Indx].fParam[1] = (*INDEX_Param_Set[0].pStepDist) * (-1.0);

								KK_Catched = 133;

								m->SeqStep++;
							}
							else
								m->SeqStep = 203;

						}

						else if(curCalib->GenSetup[SETUP_INDX_ENBL] == 1){

							if(INDEX_Param_Set[0].pStepDist){
								Process[m->pCfg->HeadCfg.INDX.PROC_Indx].xCMD = prcsSTEPpos;

								if(curCalib->GenSetup[SETUP_INDX_DIR])
									Process[m->pCfg->HeadCfg.INDX.PROC_Indx].fParam[1] = (*INDEX_Param_Set[0].pStepDist);
								else
									Process[m->pCfg->HeadCfg.INDX.PROC_Indx].fParam[1] = (*INDEX_Param_Set[0].pStepDist) * (-1.0);

								m->SeqStep++;

							}
							else
								m->SeqStep = 203;

						}
						else
							m->SeqStep = 203;

					break;

				}

			}

		break;

		case 202:

			// Always Coolant On
			if (!m->TestMode)
			{
				if (Process[m->pCfg->HeadCfg.COOL.PROC_Indx].Status != prcsSTATUS_Run)
					Process[m->pCfg->HeadCfg.COOL.PROC_Indx].xCMD = prcsSTART;
			}

			if (StopBtn)
			{
				LogTxt(&LogMgr, "Quick stop");

				m->SeqStep			= 254;			// Quick Stop
				break;
			}

			if(Process[m->pCfg->HeadCfg.INDX.PROC_Indx].Status == prcsSTATUS_Stopped
				&& Process[m->pCfg->HeadCfg.OSC.PROC_Indx].Status == prcsSTATUS_Stopped){

				TimerStart(&m->sm.Tmr1, 0.1);
				m->SeqStep++;

			}

		break;

		case 203:
			// Always Coolant On
			if (StopBtn)
			{
				LogTxt(&LogMgr, "Halt stop");

				m->SeqStep			= 254;			// Quick Stop
				break;
			}

			if (!m->TestMode)
			{
				if (Process[m->pCfg->HeadCfg.COOL.PROC_Indx].Status != prcsSTATUS_Run)
					Process[m->pCfg->HeadCfg.COOL.PROC_Indx].xCMD = prcsSTART;
			}

			if(Process[m->pCfg->HeadCfg.TVL.PROC_Indx].Status == prcsSTATUS_Stopped){

				LogTxt(&LogMgr, "M: Cyc. Time %.2f" , GlobalTimer);
				m->SeqStep++;
			}

		break;

		case 204:

			// Always Coolant On
			if (!m->TestMode)
			{
				if (Process[m->pCfg->HeadCfg.COOL.PROC_Indx].Status != prcsSTATUS_Run)
					Process[m->pCfg->HeadCfg.COOL.PROC_Indx].xCMD = prcsSTART;
			}

			ret = 5; // Preparing To Stop

			if (StopBtn)
			{
				LogTxt(&LogMgr, "Quick stop");
				m->SeqStep = 254;			// Quick Stop
				//m->SeqStep = 205;			// Normal Stop
				break;
			}

			// Check if Index move done
			if (1)
			{

				if((abs(m->curSegm[ACT_TVL_DIST] - Process[m->pCfg->HeadCfg.TVL.PROC_Indx].Param[3]) < 10)
				//if((Process[m->pCfg->HeadCfg.TVL.PROC_Indx].Status == prcsSTATUS_Stopped)
					&& (m->SubSeqStep == 2)) // IMPORTANT - head swap is only when was rewrap before
				{

					m->SubSeqStep = 1;

					//if (curCfg->Param_ENUM[parENUM_PathMode].val[0] == 0.0)
						//m->ToolHeadID = !m->ToolHeadID;

					if (curCfg->Param_ENUM[parENUM_TVL_MODE].val[0] == 0)
					{ // Relative Move
						if (TVL_ROT_Param_Set[0].pEncoder)
							OLD_MTR_POS[TVL_ENC_HOME] = *TVL_ROT_Param_Set[0].pEncoder;
					}
					AutoStartEnable = 1;
					m->SeqStep++;

				}

				else
				{
					m->SeqStep = 254;
				}

			}

		break;

		case 205:

			File_RW._int.PathDoneCnt++;
			newFile = 0;
			/*
			if (curCfg->Param_ENUM[parENUM_WeldProgramLinkMode].val[0] > 0.0)
			{

				if (curCfg->Param[parGEN_WeldProgramRepeat].val[0] == 0.0)
				{

					if (strlen(curCfg->NextProgramName) > 0)
					{

						if (!strstr(curCfg->NextProgramName, "NONE"))
						{ // Not None
							TakeNextWeldProgram(hmi);
							newFile 			= 1;

						}

					}

				}

				else
				{

					if (File_RW._int.PathDoneCnt > (UINT)curCfg->Param[parGEN_WeldProgramRepeat].val[0])
					{

						if (strlen(curCfg->NextProgramName) > 0)
						{

							if (!strstr(curCfg->NextProgramName, "NONE"))
							{ // Not None
								TakeNextWeldProgram(hmi);
								newFile 			= 1;
							}

						}

					}

				}

			}
			*/

			if (newFile)
				m->SeqStep = 206;
			else
				m->SeqStep = 207;

		break;

		case 206:
			if (File_RW.CMD == 0)
			{

				if (File_RW.Error)
					m->SeqStep = 206;

				else
				{
					AutoStartEnable = 1;
					m->SeqStep = 207;

				}
			}

		break;

		case 207:

			AutoStartEnable = 1;

			/*
			if (File_RW._int.PathDoneCnt > (UINT)curCfg->Param[parGEN_WeldProgramRepeat].val[0])
			{
				File_RW._int.PathDoneCnt = (UINT)
				curCfg->Param[parGEN_WeldProgramRepeat].val[0];

				AutoStartEnable 	= 0;
			}
			*/

			m->SeqStep++;

		break;

		case 208:
			///////////////////////////////////
			//Auto Start
			if (curCalib->GenSetup[SETUP_AUTO_START] && AutoStartEnable)
			{
				TimerStart(&m->sm.Tmr1, curCalib->GenFloatValue[SETUP_FLOAT_AUTOSTART_DLY]);
				m->SeqStep = 220;

			}
			else
				m->SeqStep = 254;

		break;

		case 210:

			if (StopBtn)
			{
				LogTxt(&LogMgr, "Quick stop");

				m->SeqStep = 254;			// Quick Stop

			}
			else if (Process[m->pCfg->HeadCfg.TVL.PROC_Indx].Status == prcsSTATUS_Stopped) // stopped by end of travel
				m->SeqStep = 0;

		break;

		case 220:

			if (StopBtn)
			{
				LogTxt(&LogMgr, "Quick stop");

				m->SeqStep = 254;			// Quick Stop
				break;
			}
			else if(!TimerIsTimeOut(&m->sm.Tmr1))
				break;

			GlobalTimer = 0;

			//WF_TVL_Diff = 0;
			LogTxt(&LogMgr, "Auto Repeat");

			if(Cont_Stop_By_End)
				AutoStartBtn = 0;
			else
				AutoStartBtn = 1;
			m->SeqStep = 0;

		break;

		case 254:

			for (i = 0; i < PROCESS_NUM; i++)
			{ // beside PROC_COOL
				if (i != PROC_COOL)
					Process[i].xCMD = prcsHalt;
			}

			Process[m->pCfg->HeadCfg.OSC.PROC_Indx].Param[0] = 1; // STop without ramp
			Process[m->pCfg->HeadCfg.OSC.PROC_Indx].xCMD = prcsQuickSTOP; // return to center position
			Process[m->pCfg->HeadCfg.GAS.PROC_Indx].xCMD = prcsSTOP; // maintain gas
			m->SeqStep++;

		break;

		default:

			if(curCfg->Param_ENUM[parENUM_AVC_Mode].val[0] != 3) // AVC Mode NOT LOCKED !
				Process[m->pCfg->HeadCfg.AVC.PROC_Indx].Param[0] = 0;

			if (StopBtn)
			{
				LogTxt(&LogMgr, "Halt stop");

				for (i = 0; i < PROCESS_NUM; i++)
				{ // beside PROC_COOL
					if (i!= PROC_COOL && i!= PROC_OSC)
						Process[i].xCMD = prcsHalt;
				}

				Process[m->pCfg->HeadCfg.GAS.PROC_Indx].xCMD = prcsSTOP; // maintain gas
				m->SeqStep			= 0;

			}

			if (Process[m->pCfg->HeadCfg.OSC.PROC_Indx].Status == prcsSTATUS_Stopped)
				m->SeqStep = 0;

			if (m->SeqStep == 0)
			{
				// Load new AVC param from new file
				TML_MTR_INST[m->pCfg->HeadCfg.AVC.TML_A_Indx]._cfg.signFilter =	curCfg->Param[parAVC_FbkFilter].val[0];
			}

		break;

		}

		//if((Process[m->pCfg->HeadCfg.TVL.PROC_Indx].Status == prcsSTATUS_Stopped))
		//StopBtn_Latch = 0;
		////////////////////////////
		TimerExecute(&WireDisable_TMR);
		TimerExecute(&WF_Catch_TMR);

		return ret;
	}

	DINT MasterSequence_Contin_OneWay(MASTER_typ * m, HMI_typ * hmi, plcbit StartBtn, plcbit StopBtn)
	{
	int 			i;
	char			status;
	DINT			ret;
	DINT			d;
	USINT			newFile;

	//Cfg_typ *cfg;
	CurCfg_typ *	curCfg;

	//CurCalib_typ *curCalib , *defCalib;
	//Scaled_Var_obj *var;
	//cfg = (Cfg_typ*) m->pCfg;
	curCfg				= (CurCfg_typ *)
	m->pCurCfg;

	//curCalib = (CurCalib_typ*) m->pCalib;
	//defCalib = (CurCalib_typ*) m->pDefaultCalib;
	//var = (Scaled_Var_obj*) m->pScaledVar;
	m->TestMode 		= intrf->TestMode;

	ret 				= 0;

	if((hmi->curHeadID == 0xFFFE)){ // Screen RUn or Alter Run

		if(intrf->GlblBtnCmd[0] &ANDR_BTN_UP){

			AVC_Param_Set[0].BoostCmd = 1;
			PS_Param_Set[0].BoostCmd = 1;
			TVL_ROT_Param_Set[0].BoostCmd = 1;
			WIRE_Param_Set[0].BoostCmd = 1;
			WIRE_Param_Set[1].BoostCmd = 1;

		}
		else if(intrf->GlblBtnCmd[0] &ANDR_BTN_DOWN){

			AVC_Param_Set[0].BoostCmd = 2;
			PS_Param_Set[0].BoostCmd = 2;
			TVL_ROT_Param_Set[0].BoostCmd = 2;
			WIRE_Param_Set[0].BoostCmd = 2;
			WIRE_Param_Set[1].BoostCmd = 2;

		}
		else{

			AVC_Param_Set[0].BoostCmd = 0;
			PS_Param_Set[0].BoostCmd = 0;
			TVL_ROT_Param_Set[0].BoostCmd = 0;
			WIRE_Param_Set[0].BoostCmd = 0;
			WIRE_Param_Set[1].BoostCmd = 0;

		}
	}
	else{

		AVC_Param_Set[0].BoostCmd = 0;
		PS_Param_Set[0].BoostCmd = 0;
		TVL_ROT_Param_Set[0].BoostCmd = 0;
		WIRE_Param_Set[0].BoostCmd = 0;
		WIRE_Param_Set[1].BoostCmd = 0;

	}

	/////////
	/////////
	//(!intrf->_intr._GlblBtnCmd[0] && (intrf->GlblBtnCmd[0] &ANDR_BTN_STOP)
	/*
	if (StopBtn)
	{
		AutoStartBtn		= 0;

		if (TimerIsTimeOut(&DoubleStop_TMR))
			TimerStart(&DoubleStop_TMR, 0.5);
		else
			DoubleStopBtn_Latch = 1;
	}

	if (StopBtn)
		StopBtn_Latch = 1;

	*/

	if (Process[m->pCfg->HeadCfg.TVL.PROC_Indx].Status != prcsSTATUS_Stopped)
	{
		if(m->SubSeqStep == 1 )// Weld to Target
		{
			//if(abs(m->curSegm[ACT_TVL_DIST] - Process[m->pCfg->HeadCfg.TVL.PROC_Indx].Param[0]) < 8){
			if(abs(m->curSegm[ACT_TVL_DIST] - Process[m->pCfg->HeadCfg.TVL.PROC_Indx].Param[0]) < 16){	// was changed July 23 2024
				m->SubSeqStep = 2;
				Weld_Report_Status = 2; // Should be reported
				LogTxt(&LogMgr, "Stopped < 1-4");
			}

			//if(abs(m->curSegm[ACT_TVL_DIST] - Process[m->pCfg->HeadCfg.TVL.PROC_Indx].Param[0]) < 10)
				//m->SubSeqStep = 2;
		}
	}

	if ((Process[m->pCfg->HeadCfg.TVL.PROC_Indx].Status == prcsSTATUS_Stopped) ||
	(Process[m->pCfg->HeadCfg.TVL.PROC_Indx].Status == prcsSTATUS_ReturnDly)){

		if(DoubleStopBtn_Latch){
			if(m->SubSeqStep > 0){
				AutoStartBtn = 0;
				m->SubSeqStep = 0;
			}
			else
				m->SubSeqStep = 1;

		}
	}
	DoubleStopBtn_Latch = 0;

	if(curCfg->Param_ENUM[parENUM_TVL_MODE].val[0] == 3) // Continues welding
		m->SubSeqStep = 0;

	if (StopBtn_Latch)
		Process[m->pCfg->HeadCfg.TVL.PROC_Indx].Param[2] = 0; // No Auto Stop and Not Rewrap

	//////////////////////////
	////////////////////////////
	if (m->SeqStep > 0)
		GlobalTimer += 0.0512; // Timer based on task class

	//////////////

		//	 MASTER SEQUENCE  //
	switch (m->SeqStep)
	{
		case 0:

			Cont_Stop_By_End = 0;
			//////////////////////////////////////
			if(curCfg->Param[parGEN_WeldProgramRepeat].val[0] == 0.0)
				File_RW._int.PathDoneCnt = 0;

			// Reset Disable when was in Test Mode
			Process[m->pCfg->HeadCfg.AVC.PROC_Indx].Disable &= 0xFD;
			Process[m->pCfg->HeadCfg.OSC.PROC_Indx].Disable &= 0xFD;
			Process[m->pCfg->HeadCfg.TVL.PROC_Indx].Disable &= 0xFD;
			Process[m->pCfg->HeadCfg.TIG.PROC_Indx].Disable &= 0xFD;
			Process[m->pCfg->HeadCfg.HW.PROC_Indx].Disable &= 0xFD;
			StopBtn_Latch = 0;

			// AVC Locked is OFF

			//if(curCfg->Param_ENUM[parENUM_AVC_Mode].val[0] != 3) // AVC Mode NOT LOCKED !
				//Process[m->pCfg->HeadCfg.AVC.PROC_Indx].Param[0] = 0;

			if(StartBtn && !Check_OSC_Amplt_and_Center())
				break;

			if (StopBtn)
			{
				LogTxt(&LogMgr, "Quick stop");
				m->SeqStep = 254;			// Halt Stop
				break;
			}

			status = 1;

			if (//(Process[m->pCfg->HeadCfg.GAS.PROC_Indx].Status != prcsSTATUS_Stopped)
				(Process[m->pCfg->HeadCfg.AVC.PROC_Indx].Status != prcsSTATUS_Stopped) ||
				(Process[m->pCfg->HeadCfg.OSC.PROC_Indx].Status != prcsSTATUS_Stopped) ||
				(Process[m->pCfg->HeadCfg.TVL.PROC_Indx].Status != prcsSTATUS_Stopped) ||
				(Process[m->pCfg->HeadCfg.WF.PROC_Indx].Status != prcsSTATUS_Stopped) ||
				(Process[m->pCfg->HeadCfg.WP.PROC_Indx].Status != prcsSTATUS_Stopped))
				status = 0;

			if (status)
			{

				if (!ErrorMgr.Error)
				{
					ret = 1;		// Raedy To Run

					if((intrf->GlblBtnCmd[0] &ANDR_BTN_HOME) && StartBtn){

						Process[m->pCfg->HeadCfg.TVL.PROC_Indx].Param[3] = 0;
						Process[m->pCfg->HeadCfg.TVL.PROC_Indx].Param[2] = 2; //only rewrap
						Process[m->pCfg->HeadCfg.TVL.PROC_Indx].xCMD = prcsSTART;
						m->SeqStep = 210;

					}

					//if ((StartBtn || AutoStartBtn) && (XMLHelper.xCmd != XML_CMD_READ))
					//if (StartBtn || AutoStartBtn)
					//else if ((StartBtn || AutoStartBtn) && ((Weld_Report_Status < 2) || ((curCalib->GenSetup[SETUP_EXTRAS]&0x1) == 0)))
					else if ((StartBtn || AutoStartBtn) && ((Weld_Report_Start_Enable) || ((curCalib->GenSetup[SETUP_EXTRAS]&0x1) == 0)))
					{
						Weld_Report_Status = 1;
						AutoStartBtn = 0;

						if (m->SubSeqStep == 2)
						{ // Rewrap

							if (curCalib->GenSetup[SETUP_SOUND_DELAY] || curCalib->GenSetup[SETUP_AUTO_START])
								TimerStart(&m->sm.Tmr1, curCalib->GenFloatValue[SETUP_FLOAT_SOUND_TM]);

							else
								TimerStart(&m->sm.Tmr1, 0.1);

							m->SeqStep = 150;

						}
						else
						{

						GlobalTimer 		= 0;

						LogTxt(&LogMgr, "PreProcess start");

						if (curCalib->GenSetup[SETUP_SOUND_DELAY] || curCalib->GenSetup[SETUP_AUTO_START])
							TimerStart(&m->sm.Tmr1, curCalib->GenFloatValue[SETUP_FLOAT_SOUND_TM]);
						else
							TimerStart(&m->sm.Tmr1, 0.1);

							m->SeqStep++;

						}
					}

					/*
					else if ((StartBtn || AutoStartBtn) && (XMLHelper.xCmd == XML_CMD_READ)){

						strcpy(hmi->pMessage[0], " FILE OPER. \n ");
						strcpy(hmi->pMessage[1], File_RW.fileName);
						strcpy(hmi->pMessage[2], "Is Loading");
						strcpy(hmi->pMessage[3] ,"Wait for finish");

						Set_Message(hmi , 0.1);

					}
					*/
				}

			}
			else
			{
				if (StopBtn)
				{
					LogTxt(&LogMgr, "Some Prcs aborted");
					m->SeqStep = 254;
				}

			}

		break;

		case 1:
		// Always Coolant On

			Cont_Stop_By_End = 0;

			if (!m->TestMode)
			{
				if (Process[m->pCfg->HeadCfg.COOL.PROC_Indx].Status != prcsSTATUS_Run)
					Process[m->pCfg->HeadCfg.COOL.PROC_Indx].xCMD = prcsSTART;
			}

			ret = 2; // Preparig To Run

			if (StopBtn)
			{
				LogTxt(&LogMgr, "Some Prcs aborted");
				m->SeqStep = 254;
			}
			else if (ErrorMgr.Error)
				m->SeqStep = 100;

			else if (!TimerIsTimeOut(&m->sm.Tmr1))
				break;

			else
			{
				if (!m->TestMode)
				{
					Process[m->pCfg->HeadCfg.GAS.PROC_Indx].xCMD = prcsSTART;
					Process[m->pCfg->HeadCfg.COOL.PROC_Indx].xCMD = prcsSTART;
				}

				if (m->TestMode)
				{

					//Process[m->pCfg->HeadCfg.AVC.PROC_Indx].Disable |= 0x02 ;
					Process[m->pCfg->HeadCfg.AVC.PROC_Indx].TestMode = 1;
					Process[m->pCfg->HeadCfg.TIG.PROC_Indx].Disable |= 0x02;
					Process[m->pCfg->HeadCfg.HW.PROC_Indx].Disable |= 0x02;

				}
				else
				{

					if ((Process[m->pCfg->HeadCfg.GAS.PROC_Indx].Status == prcsSTATUS_Run) &&
					(Process[m->pCfg->HeadCfg.COOL.PROC_Indx].Status == prcsSTATUS_Run))
					{
						//Process[m->pCfg->HeadCfg.AVC.PROC_Indx].Disable &= 0xFD ;
						Process[m->pCfg->HeadCfg.AVC.PROC_Indx].TestMode = 0;
						Process[m->pCfg->HeadCfg.TIG.PROC_Indx].Disable &= 0xFD;
						Process[m->pCfg->HeadCfg.HW.PROC_Indx].Disable &= 0xFD;

					}
					else
						break;

				}

				Process[m->pCfg->HeadCfg.AVC.PROC_Indx].xCMD = prcsSTART;

				//if(!m->TestMode)
				Process[m->pCfg->HeadCfg.TIG.PROC_Indx].xCMD = prcsForceON;

				LogTxt(&LogMgr, "ARC start");

				m->SeqStep++;

			}

		break;

		case 2:

			// Always Coolant On
			if (!m->TestMode)
			{
				if (Process[m->pCfg->HeadCfg.COOL.PROC_Indx].Status != prcsSTATUS_Run)
					Process[m->pCfg->HeadCfg.COOL.PROC_Indx].xCMD = prcsSTART;
			}

			ret = 2; // Preparig To Run

			if (StopBtn)
			{
				LogTxt(&LogMgr, "Some Prcs aborted");
				m->SeqStep			= 254;
			}

			///////////////////////////
			else if (ErrorMgr.Error)
				m->SeqStep = 100;

			else if ((Process[m->pCfg->HeadCfg.AVC.PROC_Indx].Status == prcsSTATUS_Run)
					|| (Process[m->pCfg->HeadCfg.AVC.PROC_Indx].Status == prcsSTATUS_AVC_OK))
			{

				Process[m->pCfg->HeadCfg.OSC.PROC_Indx].xCMD = prcsSTART;
				Process[m->pCfg->HeadCfg.OSC.PROC_Indx].Param[0] = 0; // Start with ramp
				Process[m->pCfg->HeadCfg.TIG.PROC_Indx].xCMD = prcsSTART;

				/*	TVL */
				Process[m->pCfg->HeadCfg.TVL.PROC_Indx].Param[2] = m->SubSeqStep;
				Process[m->pCfg->HeadCfg.TVL.PROC_Indx].xCMD = prcsSTART;

#ifdef EXTENDED_LOGS
				LogTxt(&LogMgr, "M:TVL%d Start: %.2f" , (UDINT) m->ToolHeadID , ABS_TVL_Pos);
#endif
				StartPos = 0;

				CalculateRunOverlap_Cont_OneWay();

				if (!m->WireDisabled)
				{
					// if prcsStart then Param[0] = 0 is set in Wire process - jus in case
					//Process[m->pCfg->HeadCfg.WF.PROC_Indx].Param[0] = 0; // start with full ramp
					Process[m->pCfg->HeadCfg.WF.PROC_Indx].xCMD = prcsSTART;
					//Process[m->pCfg->HeadCfg.WP.PROC_Indx].Param[0] = 0; // start with full ramp
					Process[m->pCfg->HeadCfg.WP.PROC_Indx].xCMD = prcsSTART;
					Process[m->pCfg->HeadCfg.HW.PROC_Indx].xCMD = prcsSTART;
				}

				LogTxt(&LogMgr, "ARC established");

				TimerStart(&WireDisable_TMR, 3.0);

				m->SeqStep++;

			}

		break;

		case 3:
			// Always Coolant On
			if (!m->TestMode)
			{
				if (Process[m->pCfg->HeadCfg.COOL.PROC_Indx].Status != prcsSTATUS_Run)
					Process[m->pCfg->HeadCfg.COOL.PROC_Indx].xCMD = prcsSTART;
			}

			WireDisableInable(WireDisable_TMR.Q);
			Process[m->pCfg->HeadCfg.TIG.PROC_Indx].Param[0] = Process[m->pCfg->HeadCfg.OSC.PROC_Indx].subStatus;
			Process[m->pCfg->HeadCfg.HW.PROC_Indx].Param[0] = Process[m->pCfg->HeadCfg.OSC.PROC_Indx].subStatus;
			ret = 3; //  Run

			//if (actRot != _actRot)
				//TakeNextWeldProgram(hmi);

			_actRot = actRot;

			if (Process[m->pCfg->HeadCfg.TVL.PROC_Indx].subStatus == 1)
			{ // End of travel reached
				//LogTxt(&LogMgr, "Path Done");
				//LogTxt(&LogMgr, "Path Done: %.2f" , ABS_TVL_Pos);

				Weld_Report_Status = 2;

				m->SeqStep = 200;

			}

			if (StopBtn)		{

				/*
				LogTxt(&LogMgr, "Process stop");
				//Process[m->pCfg->HeadCfg.TVL.PROC_Indx].xCMD = prcsSTOP;
				m->SeqStep = 200;
				*/
				if(Cont_Stop_By_End){
					LogTxt(&LogMgr, "Process stop by Operator");
					Cont_Stop_By_End = 0;
					m->SeqStep = 200;
				}
				else
					Cont_Stop_By_End = 1;

			}
			else if (ErrorMgr.Error || m->ESTOP)
			{
				LogTxt(&LogMgr, "Process Error");
				m->SeqStep = 100;
			}

		break;

		case 100:
			// Always Coolant On
			if (!m->TestMode)
			{
				if (Process[m->pCfg->HeadCfg.COOL.PROC_Indx].Status != prcsSTATUS_Run)
					Process[m->pCfg->HeadCfg.COOL.PROC_Indx].xCMD = prcsSTART;
			}

			Process[m->pCfg->HeadCfg.TVL.PROC_Indx].xCMD = prcsHalt;
			Process[m->pCfg->HeadCfg.OSC.PROC_Indx].xCMD = prcsHalt;
			Process[m->pCfg->HeadCfg.AVC.PROC_Indx].xCMD = prcsHalt;
			Process[m->pCfg->HeadCfg.WF.PROC_Indx].xCMD = prcsHalt;
			Process[m->pCfg->HeadCfg.WP.PROC_Indx].xCMD = prcsHalt;
			Process[m->pCfg->HeadCfg.TIG.PROC_Indx].xCMD = prcsHalt;
			Process[m->pCfg->HeadCfg.HW.PROC_Indx].xCMD = prcsHalt;
			Process[m->pCfg->HeadCfg.GAS.PROC_Indx].xCMD = prcsSTOP;

			//Process[m->pCfg->HeadCfg.COOL.PROC_Indx].xCMD = prcsHalt;
			switch (ErrorMgr.Error)
			{
				case ERROR_FATAL:
					m->SeqStep++;
				break;

				case ERROR_MOTOR:
					m->SeqStep++;
				break;

				case ERROR_MOTOR_INIT:
					m->SeqStep++;
				break;

				case ERROR_TIG_PROC:
					m->SeqStep++;
				break;

				default:
					m->SeqStep++;
				break;
			}

		break;

		case 101:
			ret = 4; // Preparig To Stop in Halt Mode

			if (StopBtn)
			{
				for (i = 0; i < PROCESS_NUM; i++)
				{
					if (i != PROC_COOL)
						Process[i].xCMD = prcsHalt;
				}
				Process[m->pCfg->HeadCfg.GAS.PROC_Indx].xCMD = prcsSTOP; // maintain gas
			}

			status = 1;

			if (Process[m->pCfg->HeadCfg.TVL.PROC_Indx].Status != prcsSTATUS_Stopped)
				status = 0;

			if (Process[m->pCfg->HeadCfg.OSC.PROC_Indx].Status != prcsSTATUS_Stopped)
				status = 0;

			if (Process[m->pCfg->HeadCfg.AVC.PROC_Indx].Status != prcsSTATUS_Stopped)
				status = 0;

			if (Process[m->pCfg->HeadCfg.WF.PROC_Indx].Status != prcsSTATUS_Stopped)
				status = 0;

			if (Process[m->pCfg->HeadCfg.GAS.PROC_Indx].Status != prcsSTATUS_Stopped)
				status = 0;

			if (Process[m->pCfg->HeadCfg.WP.PROC_Indx].Status != prcsSTATUS_Stopped)
				status = 0;

			if (Process[m->pCfg->HeadCfg.TIG.PROC_Indx].Status != prcsSTATUS_Stopped)
				status = 0;

			if (Process[m->pCfg->HeadCfg.HW.PROC_Indx].Status != prcsSTATUS_Stopped)
				status = 0;

			if (status)
			{
				LogTxt(&LogMgr, "Prc Final stopped");
				m->SeqStep = 254;
			}

		break;

		case 150:

			if (StopBtn)
			{
				LogTxt(&LogMgr, "Quick stop");
				m->SeqStep = 254;			// Quick Stop
				break;
			}

			if (!TimerIsTimeOut(&m->sm.Tmr1))
				break;

			/*	TVL */
			Process[m->pCfg->HeadCfg.TVL.PROC_Indx].Param[2] = m->SubSeqStep;
			Process[m->pCfg->HeadCfg.TVL.PROC_Indx].xCMD = prcsSTART;
			StartPos = 0;

			CalculateRunOverlap_Cont_OneWay();

			m->SeqStep = 202;

		break;

		case 200:

			// Always Coolant On
			if (!m->TestMode)
			{
				if (Process[m->pCfg->HeadCfg.COOL.PROC_Indx].Status != prcsSTATUS_Run)
					Process[m->pCfg->HeadCfg.COOL.PROC_Indx].xCMD = prcsSTART;
			}

			for (i = 0; i < PROCESS_NUM; i++)
			{
				if((i != PROC_COOL))
					//&&( i != m->pCfg->HeadCfg.TVL.PROC_Indx))
					Process[i].xCMD = prcsSTOP;

			}

			// Dodane - Nie ma Xcmd Stop w TRVL_BPV_POS
			if((TVL_ROT_Param_Set[0].Mode == 2) // with only position
				|| (TVL_ROT_Param_Set[0].Mode == 3)) // with interrupt
				Process[m->pCfg->HeadCfg.TVL.PROC_Indx].xCMD = 0;

///////////////////////////////////////////////////////////////////////////
/// Nowosc Index wczesniej

			if((curCalib->GenSetup[SETUP_EXTRAS]&0x4)){

				switch(curCalib->GenSetup[SETUP_HEAD_SETUP] ){

						default:

							if(curCalib->GenSetup[SETUP_INDX_ENBL] == 3){ // In OSc

								if(INDEX_Param_Set[0].pStepDist){

									Process[m->pCfg->HeadCfg.OSC.PROC_Indx].xCMD = prcsSTEPneg; // Quick Step with delay

									if(curCalib->GenSetup[SETUP_INDX_DIR])
										Process[m->pCfg->HeadCfg.OSC.PROC_Indx].fParam[1] = (*INDEX_Param_Set[0].pStepDist);
									else
										Process[m->pCfg->HeadCfg.OSC.PROC_Indx].fParam[1] = (*INDEX_Param_Set[0].pStepDist) * (-1.0);

									KK_Catched = 133;

									//m->SeqStep++;
								}
								//else
									//m->SeqStep = 203;

							}

							else if(curCalib->GenSetup[SETUP_INDX_ENBL] == 1){

								if(INDEX_Param_Set[0].pStepDist){
									Process[m->pCfg->HeadCfg.INDX.PROC_Indx].xCMD = prcsSTEPpos;

									if(curCalib->GenSetup[SETUP_INDX_DIR])
										Process[m->pCfg->HeadCfg.INDX.PROC_Indx].fParam[1] = (*INDEX_Param_Set[0].pStepDist);
									else
										Process[m->pCfg->HeadCfg.INDX.PROC_Indx].fParam[1] = (*INDEX_Param_Set[0].pStepDist) * (-1.0);

									m->SeqStep++;

								}
								//else
									//m->SeqStep = 203;

							}
							//else
								//m->SeqStep = 203;

						break;

					}

			}

/////////////////////////////////////////////////////////////////////////
/////////////////////////////////////////////////////////////////////////
#ifdef EXTENDED_LOGS

			LogTxt(&LogMgr, "Path %d Done: %.2f" , (UDINT)File_RW._int.PathDoneCnt, ABS_TVL_Pos);
#else
			LogTxt(&LogMgr, "Path %d Done" , (UDINT)File_RW._int.PathDoneCnt);

#endif

			//TimerStart(&WF_Catch_TMR, curCfg->Param[parWF_RampDwn].val[0]);
			m->SeqStep++;

		break;

		case 201:

			// Always Coolant On
			if (!m->TestMode)
			{
				if (Process[m->pCfg->HeadCfg.COOL.PROC_Indx].Status != prcsSTATUS_Run)
					Process[m->pCfg->HeadCfg.COOL.PROC_Indx].xCMD = prcsSTART;
			}

			ret = 5; // Preparing To Stop

			if (StopBtn)
			{
#ifdef EXTENDED_LOGS

				LogTxt(&LogMgr, "Quick stop %.2f" , ABS_TVL_Pos);
#else
				LogTxt(&LogMgr, "Quick stop");
#endif
				m->SeqStep = 254;			// Quick Stop
			}

			status = 1;

			if (Process[m->pCfg->HeadCfg.TVL.PROC_Indx].Status != prcsSTATUS_Stopped){ // stopped by end of travel
				status = 0;
			}

			if (Process[m->pCfg->HeadCfg.INDX.PROC_Indx].Status != prcsSTATUS_Stopped){
				status = 0;
			}

			if (Process[m->pCfg->HeadCfg.OSC.PROC_Indx].Status != prcsSTATUS_Stopped)
				status = 0;

			if (Process[m->pCfg->HeadCfg.AVC.PROC_Indx].Status != prcsSTATUS_Stopped)
				status = 0;

			if (Process[m->pCfg->HeadCfg.WF.PROC_Indx].Status != prcsSTATUS_Stopped)
				status = 0;

			//if (Process[m->pCfg->HeadCfg.GAS.PROC_Indx].Status != prcsSTATUS_Stopped)
				//status = 0;

			if (Process[m->pCfg->HeadCfg.WP.PROC_Indx].Status != prcsSTATUS_Stopped)
				status = 0;

			if (Process[m->pCfg->HeadCfg.TIG.PROC_Indx].Status != prcsSTATUS_Stopped)
				status = 0;

			if (Process[m->pCfg->HeadCfg.HW.PROC_Indx].Status != prcsSTATUS_Stopped)
				status = 0;

			if (status)
			{

#ifdef EXTENDED_LOGS

				LogTxt(&LogMgr, "M:All%d Stop: %.2f" ,(UDINT) m->ToolHeadID, ABS_TVL_Pos);

#endif
				if(!(curCalib->GenSetup[SETUP_EXTRAS]&0x4)){

					switch(curCalib->GenSetup[SETUP_HEAD_SETUP] ){

						default:

							if(curCalib->GenSetup[SETUP_INDX_ENBL] == 3){ // In OSc

								if(INDEX_Param_Set[0].pStepDist){

									Process[m->pCfg->HeadCfg.OSC.PROC_Indx].xCMD = prcsSTEPpos;

									if(curCalib->GenSetup[SETUP_INDX_DIR])
										Process[m->pCfg->HeadCfg.OSC.PROC_Indx].fParam[1] = (*INDEX_Param_Set[0].pStepDist);
									else
										Process[m->pCfg->HeadCfg.OSC.PROC_Indx].fParam[1] = (*INDEX_Param_Set[0].pStepDist) * (-1.0);

									KK_Catched = 133;

									m->SeqStep++;
								}
								else
									m->SeqStep = 203;

							}

							else if(curCalib->GenSetup[SETUP_INDX_ENBL] == 1){

								if(INDEX_Param_Set[0].pStepDist){
									Process[m->pCfg->HeadCfg.INDX.PROC_Indx].xCMD = prcsSTEPpos;

									if(curCalib->GenSetup[SETUP_INDX_DIR])
										Process[m->pCfg->HeadCfg.INDX.PROC_Indx].fParam[1] = (*INDEX_Param_Set[0].pStepDist);
									else
										Process[m->pCfg->HeadCfg.INDX.PROC_Indx].fParam[1] = (*INDEX_Param_Set[0].pStepDist) * (-1.0);

									m->SeqStep++;

								}
								else
									m->SeqStep = 203;

							}
							else
								m->SeqStep = 203;

						break;

					}
					}

				m->SeqStep++;

			}

		break;

		case 202:

			// Always Coolant On
			if (!m->TestMode)
			{
				if (Process[m->pCfg->HeadCfg.COOL.PROC_Indx].Status != prcsSTATUS_Run)
					Process[m->pCfg->HeadCfg.COOL.PROC_Indx].xCMD = prcsSTART;
			}

			if (StopBtn)
			{
				LogTxt(&LogMgr, "Quick stop");

				m->SeqStep			= 254;			// Quick Stop
				break;
			}

			if(Process[m->pCfg->HeadCfg.INDX.PROC_Indx].Status == prcsSTATUS_Stopped
				&& Process[m->pCfg->HeadCfg.OSC.PROC_Indx].Status == prcsSTATUS_Stopped){

				TimerStart(&m->sm.Tmr1, 0.1);
				m->SeqStep++;

			}

		break;

		case 203:
			// Always Coolant On
			if (StopBtn)
			{
				LogTxt(&LogMgr, "Halt stop");

				m->SeqStep			= 254;			// Quick Stop
				break;
			}

			if (!m->TestMode)
			{
				if (Process[m->pCfg->HeadCfg.COOL.PROC_Indx].Status != prcsSTATUS_Run)
					Process[m->pCfg->HeadCfg.COOL.PROC_Indx].xCMD = prcsSTART;
			}

			if(Process[m->pCfg->HeadCfg.TVL.PROC_Indx].Status == prcsSTATUS_Stopped){

				LogTxt(&LogMgr, "M: Cyc. Time %.2f" , GlobalTimer);
				m->SeqStep++;
			}

		break;

		case 204:

			// Always Coolant On
			if (!m->TestMode)
			{
				if (Process[m->pCfg->HeadCfg.COOL.PROC_Indx].Status != prcsSTATUS_Run)
					Process[m->pCfg->HeadCfg.COOL.PROC_Indx].xCMD = prcsSTART;
			}

			ret = 5; // Preparing To Stop

			if (StopBtn)
			{
				LogTxt(&LogMgr, "Quick stop");
				m->SeqStep = 254;			// Quick Stop
				//m->SeqStep = 205;			// Normal Stop
				break;
			}

			// Check if Index move done
			if (1)
			{

				if((abs(m->curSegm[ACT_TVL_DIST] - Process[m->pCfg->HeadCfg.TVL.PROC_Indx].Param[3]) < 10)
				//if((Process[m->pCfg->HeadCfg.TVL.PROC_Indx].Status == prcsSTATUS_Stopped)
					&& (m->SubSeqStep == 2)) // IMPORTANT - head swap is only when was rewrap before
				{

					m->SubSeqStep = 1;

					//if (curCfg->Param_ENUM[parENUM_PathMode].val[0] == 0.0)
						//m->ToolHeadID = !m->ToolHeadID;

					if (curCfg->Param_ENUM[parENUM_TVL_MODE].val[0] == 0)
					{ // Relative Move
						if (TVL_ROT_Param_Set[0].pEncoder)
							OLD_MTR_POS[TVL_ENC_HOME] = *TVL_ROT_Param_Set[0].pEncoder;
					}
					AutoStartEnable = 1;
					m->SeqStep++;

				}

				else
				{
					m->SeqStep = 254;
				}

			}

		break;

		case 205:

			File_RW._int.PathDoneCnt++;
			newFile = 0;
			/*
			if (curCfg->Param_ENUM[parENUM_WeldProgramLinkMode].val[0] > 0.0)
			{

				if (curCfg->Param[parGEN_WeldProgramRepeat].val[0] == 0.0)
				{

					if (strlen(curCfg->NextProgramName) > 0)
					{

						if (!strstr(curCfg->NextProgramName, "NONE"))
						{ // Not None
							TakeNextWeldProgram(hmi);
							newFile 			= 1;

						}

					}

				}

				else
				{

					if (File_RW._int.PathDoneCnt > (UINT)curCfg->Param[parGEN_WeldProgramRepeat].val[0])
					{

						if (strlen(curCfg->NextProgramName) > 0)
						{

							if (!strstr(curCfg->NextProgramName, "NONE"))
							{ // Not None
								TakeNextWeldProgram(hmi);
								newFile 			= 1;
							}

						}

					}

				}

			}
			*/

			if (newFile)
				m->SeqStep = 206;
			else
				m->SeqStep = 207;

		break;

		case 206:
			if (File_RW.CMD == 0)
			{

				if (File_RW.Error)
					m->SeqStep = 206;

				else
				{
					AutoStartEnable = 1;
					m->SeqStep = 207;

				}
			}

		break;

		case 207:

			AutoStartEnable = 1;

			/*
			if (File_RW._int.PathDoneCnt > (UINT)curCfg->Param[parGEN_WeldProgramRepeat].val[0])
			{
				File_RW._int.PathDoneCnt = (UINT)
				curCfg->Param[parGEN_WeldProgramRepeat].val[0];

				AutoStartEnable 	= 0;
			}
			*/

			m->SeqStep++;

		break;

		case 208:
			///////////////////////////////////
			//Auto Start
			if (curCalib->GenSetup[SETUP_AUTO_START] && AutoStartEnable)
			{
				TimerStart(&m->sm.Tmr1, curCalib->GenFloatValue[SETUP_FLOAT_AUTOSTART_DLY]);
				m->SeqStep = 220;

			}
			else
				m->SeqStep = 254;

		break;

		case 210:

			if (StopBtn)
			{
				LogTxt(&LogMgr, "Quick stop");

				m->SeqStep = 254;			// Quick Stop

			}
			else if (Process[m->pCfg->HeadCfg.TVL.PROC_Indx].Status == prcsSTATUS_Stopped) // stopped by end of travel
				m->SeqStep = 0;

		break;

		case 220:

			if (StopBtn)
			{
				LogTxt(&LogMgr, "Quick stop");

				m->SeqStep = 254;			// Quick Stop
				break;
			}
			else if(!TimerIsTimeOut(&m->sm.Tmr1))
				break;

			GlobalTimer = 0;

			//WF_TVL_Diff = 0;
			LogTxt(&LogMgr, "Auto Repeat");

			if(Cont_Stop_By_End)
				AutoStartBtn = 0;
			else
				AutoStartBtn = 1;
			m->SeqStep = 0;

		break;

		case 254:

			for (i = 0; i < PROCESS_NUM; i++)
			{ // beside PROC_COOL
				if (i != PROC_COOL)
					Process[i].xCMD = prcsHalt;
			}

			Process[m->pCfg->HeadCfg.OSC.PROC_Indx].Param[0] = 1; // STop without ramp
			Process[m->pCfg->HeadCfg.OSC.PROC_Indx].xCMD = prcsQuickSTOP; // return to center position
			Process[m->pCfg->HeadCfg.GAS.PROC_Indx].xCMD = prcsSTOP; // maintain gas
			m->SeqStep++;

		break;

		default:

			if(curCfg->Param_ENUM[parENUM_AVC_Mode].val[0] != 3) // AVC Mode NOT LOCKED !
				Process[m->pCfg->HeadCfg.AVC.PROC_Indx].Param[0] = 0;

			if (StopBtn)
			{
				LogTxt(&LogMgr, "Halt stop");

				for (i = 0; i < PROCESS_NUM; i++)
				{ // beside PROC_COOL
					if (i!= PROC_COOL && i!= PROC_OSC)
						Process[i].xCMD = prcsHalt;
				}

				Process[m->pCfg->HeadCfg.GAS.PROC_Indx].xCMD = prcsSTOP; // maintain gas
				m->SeqStep			= 0;

			}

			if (Process[m->pCfg->HeadCfg.OSC.PROC_Indx].Status == prcsSTATUS_Stopped)
				m->SeqStep = 0;

			if (m->SeqStep == 0)
			{
				// Load new AVC param from new file
				TML_MTR_INST[m->pCfg->HeadCfg.AVC.TML_A_Indx]._cfg.signFilter =	curCfg->Param[parAVC_FbkFilter].val[0];
			}

		break;

		}

		//if((Process[m->pCfg->HeadCfg.TVL.PROC_Indx].Status == prcsSTATUS_Stopped))
		//StopBtn_Latch = 0;
		////////////////////////////
		TimerExecute(&WireDisable_TMR);
		TimerExecute(&WF_Catch_TMR);

		return ret;
	}

	DINT MasterSequence_Contin(MASTER_typ * m, HMI_typ * hmi, plcbit StartBtn, plcbit StopBtn)
	{
	int 			i;
	char			status;
	DINT			ret;
	DINT			d;
	USINT			newFile;

	//Cfg_typ *cfg;
	CurCfg_typ *	curCfg;

	//CurCalib_typ *curCalib , *defCalib;
	//Scaled_Var_obj *var;
	//cfg = (Cfg_typ*) m->pCfg;
	curCfg				= (CurCfg_typ *)
	m->pCurCfg;

	//curCalib = (CurCalib_typ*) m->pCalib;
	//defCalib = (CurCalib_typ*) m->pDefaultCalib;
	//var = (Scaled_Var_obj*) m->pScaledVar;
	m->TestMode 		= intrf->TestMode;

	ret 				= 0;

	if((hmi->curHeadID == 0xFFFE)){ // Screen RUn or Alter Run

		if(intrf->GlblBtnCmd[0] &ANDR_BTN_UP){

			AVC_Param_Set[0].BoostCmd = 1;
			PS_Param_Set[0].BoostCmd = 1;
			TVL_ROT_Param_Set[0].BoostCmd = 1;
			WIRE_Param_Set[0].BoostCmd = 1;
			WIRE_Param_Set[1].BoostCmd = 1;

		}
		else if(intrf->GlblBtnCmd[0] &ANDR_BTN_DOWN){

			AVC_Param_Set[0].BoostCmd = 2;
			PS_Param_Set[0].BoostCmd = 2;
			TVL_ROT_Param_Set[0].BoostCmd = 2;
			WIRE_Param_Set[0].BoostCmd = 2;
			WIRE_Param_Set[1].BoostCmd = 2;

		}
		else{

			AVC_Param_Set[0].BoostCmd = 0;
			PS_Param_Set[0].BoostCmd = 0;
			TVL_ROT_Param_Set[0].BoostCmd = 0;
			WIRE_Param_Set[0].BoostCmd = 0;
			WIRE_Param_Set[1].BoostCmd = 0;

		}
	}
	else{

		AVC_Param_Set[0].BoostCmd = 0;
		PS_Param_Set[0].BoostCmd = 0;
		TVL_ROT_Param_Set[0].BoostCmd = 0;
		WIRE_Param_Set[0].BoostCmd = 0;
		WIRE_Param_Set[1].BoostCmd = 0;

	}

	/////////
	if (StopBtn)
	{
		AutoStartBtn		= 0;

		if (TimerIsTimeOut(&DoubleStop_TMR))
			TimerStart(&DoubleStop_TMR, 0.5);
		else
			DoubleStopBtn_Latch = 1;
	}

	if (StopBtn)
		StopBtn_Latch = 1;

	m->SubSeqStep = 3; // Only Information that target is reached

	/*
	if ((Process[m->pCfg->HeadCfg.TVL.PROC_Indx].Status == prcsSTATUS_Stopped) ||
	(Process[m->pCfg->HeadCfg.TVL.PROC_Indx].Status == prcsSTATUS_ReturnDly)){

		if (DoubleStopBtn_Latch)
			m->SubSeqStep = 0;
	}
	DoubleStopBtn_Latch = 0;

	if(curCfg->Param_ENUM[parENUM_TVL_MODE].val[0] == 3) // Continues welding
		m->SubSeqStep = 0;

	if (StopBtn_Latch)
		Process[m->pCfg->HeadCfg.TVL.PROC_Indx].Param[2] = 0; // No Auto Stop and Not Rewrap

	*/

	//////////////////////////
	////////////////////////////
	if (m->SeqStep > 0)
		GlobalTimer += 0.0512; // Timer based on task class

	//////////////

		//	 MASTER SEQUENCE  //
	switch (m->SeqStep)
	{
		case 0:

			Cont_Stop_By_End = 0;
			Process[m->pCfg->HeadCfg.AVC.PROC_Indx].Param[0] = 0; // AVC UnLocked

			//////////////////////////////////////
			if(curCfg->Param[parGEN_WeldProgramRepeat].val[0] == 0.0)
				File_RW._int.PathDoneCnt = 0;

			// Reset Disable when was in Test Mode
			Process[m->pCfg->HeadCfg.AVC.PROC_Indx].Disable &= 0xFD;
			Process[m->pCfg->HeadCfg.OSC.PROC_Indx].Disable &= 0xFD;
			Process[m->pCfg->HeadCfg.TVL.PROC_Indx].Disable &= 0xFD;
			Process[m->pCfg->HeadCfg.TIG.PROC_Indx].Disable &= 0xFD;
			Process[m->pCfg->HeadCfg.HW.PROC_Indx].Disable &= 0xFD;
			StopBtn_Latch = 0;

			// AVC Locked is OFF

			//if(curCfg->Param_ENUM[parENUM_AVC_Mode].val[0] != 3) // AVC Mode NOT LOCKED !
				//Process[m->pCfg->HeadCfg.AVC.PROC_Indx].Param[0] = 0;

			if(StartBtn && !Check_OSC_Amplt_and_Center())
				break;

			if (StopBtn)
			{
				LogTxt(&LogMgr, "Quick stop");
				m->SeqStep = 254;			// Halt Stop
				break;
			}

			status = 1;

			if (//(Process[m->pCfg->HeadCfg.GAS.PROC_Indx].Status != prcsSTATUS_Stopped)
				(Process[m->pCfg->HeadCfg.AVC.PROC_Indx].Status != prcsSTATUS_Stopped) ||
				(Process[m->pCfg->HeadCfg.OSC.PROC_Indx].Status != prcsSTATUS_Stopped) ||
				(Process[m->pCfg->HeadCfg.TVL.PROC_Indx].Status != prcsSTATUS_Stopped) ||
				(Process[m->pCfg->HeadCfg.WF.PROC_Indx].Status != prcsSTATUS_Stopped) ||
				(Process[m->pCfg->HeadCfg.WP.PROC_Indx].Status != prcsSTATUS_Stopped))
				status = 0;

			if (status)
			{

				if (!ErrorMgr.Error)
				{
					ret = 1;		// Raedy To Run

					if (StartBtn)
					//if (StartBtn || AutoStartBtn)
					{

						AutoStartBtn = 0;

						GlobalTimer 		= 0;

						LogTxt(&LogMgr, "PreProcess start");

						if (curCalib->GenSetup[SETUP_SOUND_DELAY] || curCalib->GenSetup[SETUP_AUTO_START])
							TimerStart(&m->sm.Tmr1, curCalib->GenFloatValue[SETUP_FLOAT_SOUND_TM]);
						else
							TimerStart(&m->sm.Tmr1, 0.1);

						m->SeqStep++;

					}
				}

			}
			else
			{
				if (StopBtn)
				{
					LogTxt(&LogMgr, "Some Prcs aborted");
					m->SeqStep = 254;
				}

			}

		break;

		case 1:

			Cont_Stop_By_End = 0;
		// Always Coolant On
			if (!m->TestMode)
			{
				if (Process[m->pCfg->HeadCfg.COOL.PROC_Indx].Status != prcsSTATUS_Run)
					Process[m->pCfg->HeadCfg.COOL.PROC_Indx].xCMD = prcsSTART;
			}

			ret = 2; // Preparig To Run

			if (StopBtn)
			{
				LogTxt(&LogMgr, "Some Prcs aborted");
				m->SeqStep = 254;
			}
			else if (ErrorMgr.Error)
				m->SeqStep = 100;

			else if (!TimerIsTimeOut(&m->sm.Tmr1))
				break;

			else
			{

				/*
				if (!m->TestMode)
				{
					Process[m->pCfg->HeadCfg.GAS.PROC_Indx].xCMD = prcsSTART;
					Process[m->pCfg->HeadCfg.COOL.PROC_Indx].xCMD = prcsSTART;
				}
				*/

				if (m->TestMode)
				{

					//Process[m->pCfg->HeadCfg.AVC.PROC_Indx].Disable |= 0x02 ;
					Process[m->pCfg->HeadCfg.AVC.PROC_Indx].TestMode = 1;
					Process[m->pCfg->HeadCfg.TIG.PROC_Indx].Disable |= 0x02;
					Process[m->pCfg->HeadCfg.HW.PROC_Indx].Disable |= 0x02;

				}
				else
				{

					Process[m->pCfg->HeadCfg.GAS.PROC_Indx].xCMD = prcsSTART;
					Process[m->pCfg->HeadCfg.COOL.PROC_Indx].xCMD = prcsSTART;

					if ((Process[m->pCfg->HeadCfg.GAS.PROC_Indx].Status == prcsSTATUS_Run) &&
					(Process[m->pCfg->HeadCfg.COOL.PROC_Indx].Status == prcsSTATUS_Run))
					{
						//Process[m->pCfg->HeadCfg.AVC.PROC_Indx].Disable &= 0xFD ;
						Process[m->pCfg->HeadCfg.AVC.PROC_Indx].TestMode = 0;
						Process[m->pCfg->HeadCfg.TIG.PROC_Indx].Disable &= 0xFD;
						Process[m->pCfg->HeadCfg.HW.PROC_Indx].Disable &= 0xFD;

					}
					else
						break;

				}

				Process[m->pCfg->HeadCfg.AVC.PROC_Indx].xCMD = prcsSTART;

				//if(!m->TestMode)
				Process[m->pCfg->HeadCfg.TIG.PROC_Indx].xCMD = prcsForceON;

				LogTxt(&LogMgr, "ARC start");

				m->SeqStep++;

			}

		break;

		case 2:

			// Always Coolant On
			if (!m->TestMode)
			{
				if (Process[m->pCfg->HeadCfg.COOL.PROC_Indx].Status != prcsSTATUS_Run)
					Process[m->pCfg->HeadCfg.COOL.PROC_Indx].xCMD = prcsSTART;
			}

			ret = 2; // Preparig To Run

			if (StopBtn)
			{
				LogTxt(&LogMgr, "Some Prcs aborted");
				m->SeqStep			= 254;
			}

			///////////////////////////
			else if (ErrorMgr.Error)
				m->SeqStep = 100;

			else if ((Process[m->pCfg->HeadCfg.AVC.PROC_Indx].Status == prcsSTATUS_Run)
					|| (Process[m->pCfg->HeadCfg.AVC.PROC_Indx].Status == prcsSTATUS_AVC_OK))
			{

				Process[m->pCfg->HeadCfg.OSC.PROC_Indx].xCMD = prcsSTART;
				Process[m->pCfg->HeadCfg.OSC.PROC_Indx].Param[0] = 0; // Start with ramp
				Process[m->pCfg->HeadCfg.TIG.PROC_Indx].xCMD = prcsSTART;

				/*	TVL */
				Process[m->pCfg->HeadCfg.TVL.PROC_Indx].Param[2] = m->SubSeqStep;

				Process[m->pCfg->HeadCfg.TVL.PROC_Indx].xCMD = prcsSTART;

#ifdef EXTENDED_LOGS
				LogTxt(&LogMgr, "M:TVL%d Start: %.2f" , (UDINT) m->ToolHeadID , ABS_TVL_Pos);
#endif
				StartPos = 0;

				CalculateRunOverlap_Cont();

				if (!m->WireDisabled)
				{
					Process[m->pCfg->HeadCfg.WF.PROC_Indx].xCMD = prcsSTART;
					Process[m->pCfg->HeadCfg.WP.PROC_Indx].xCMD = prcsSTART;
					Process[m->pCfg->HeadCfg.HW.PROC_Indx].xCMD = prcsSTART;
				}

				LogTxt(&LogMgr, "ARC established");

				TimerStart(&WireDisable_TMR, 3.0);

				m->SeqStep++;

			}

		break;

		case 3:
			// Always Coolant On
			if (!m->TestMode)
			{
				if (Process[m->pCfg->HeadCfg.COOL.PROC_Indx].Status != prcsSTATUS_Run)
					Process[m->pCfg->HeadCfg.COOL.PROC_Indx].xCMD = prcsSTART;
			}

			WireDisableInable(WireDisable_TMR.Q);
			Process[m->pCfg->HeadCfg.TIG.PROC_Indx].Param[0] = Process[m->pCfg->HeadCfg.OSC.PROC_Indx].subStatus;
			Process[m->pCfg->HeadCfg.HW.PROC_Indx].Param[0] = Process[m->pCfg->HeadCfg.OSC.PROC_Indx].subStatus;
			ret = 3; //  Run

			/*
			if (actRot != _actRot)
				TakeNextWeldProgram(hmi);
			*/
			_actRot = actRot;

			if (Process[m->pCfg->HeadCfg.TVL.PROC_Indx].subStatus == 1)
			{
				if(Cont_Stop_By_End){

					m->SeqStep = 240; // Regular Stop
				}
				else{

					m->SeqStep = 200;

				}

			}

			if (StopBtn) // Stop by operator
			{
				if(Cont_Stop_By_End){
					LogTxt(&LogMgr, "Process stop by Operator");
					Cont_Stop_By_End = 0;
					m->SeqStep = 240;
				}
				else
					Cont_Stop_By_End = 1;

			}
			else if (ErrorMgr.Error || m->ESTOP)
			{
				LogTxt(&LogMgr, "Process Error");
				m->SeqStep = 100;
			}

		break;

		case 100:
			// Always Coolant On
			if (!m->TestMode)
			{
				if (Process[m->pCfg->HeadCfg.COOL.PROC_Indx].Status != prcsSTATUS_Run)
					Process[m->pCfg->HeadCfg.COOL.PROC_Indx].xCMD = prcsSTART;
			}

			Process[m->pCfg->HeadCfg.TVL.PROC_Indx].xCMD = prcsHalt;
			Process[m->pCfg->HeadCfg.OSC.PROC_Indx].xCMD = prcsHalt;
			Process[m->pCfg->HeadCfg.AVC.PROC_Indx].xCMD = prcsHalt;
			Process[m->pCfg->HeadCfg.WF.PROC_Indx].xCMD = prcsHalt;
			Process[m->pCfg->HeadCfg.WP.PROC_Indx].xCMD = prcsHalt;
			Process[m->pCfg->HeadCfg.TIG.PROC_Indx].xCMD = prcsHalt;
			Process[m->pCfg->HeadCfg.HW.PROC_Indx].xCMD = prcsHalt;
			Process[m->pCfg->HeadCfg.GAS.PROC_Indx].xCMD = prcsSTOP;

			//Process[m->pCfg->HeadCfg.COOL.PROC_Indx].xCMD = prcsHalt;
			switch (ErrorMgr.Error)
			{
				case ERROR_FATAL:
					m->SeqStep++;
				break;

				case ERROR_MOTOR:
					m->SeqStep++;
				break;

				case ERROR_MOTOR_INIT:
					m->SeqStep++;
				break;

				case ERROR_TIG_PROC:
					m->SeqStep++;
				break;

				default:
					m->SeqStep++;
				break;
			}

		break;

		case 101:
			ret = 4; // Preparig To Stop in Halt Mode

			if (StopBtn)
			{
				for (i = 0; i < PROCESS_NUM; i++)
				{
					if (i != PROC_COOL)
						Process[i].xCMD = prcsHalt;
				}
				Process[m->pCfg->HeadCfg.GAS.PROC_Indx].xCMD = prcsSTOP; // maintain gas
			}

			status = 1;

			if (Process[m->pCfg->HeadCfg.TVL.PROC_Indx].Status != prcsSTATUS_Stopped)
				status = 0;

			if (Process[m->pCfg->HeadCfg.OSC.PROC_Indx].Status != prcsSTATUS_Stopped)
				status = 0;

			if (Process[m->pCfg->HeadCfg.AVC.PROC_Indx].Status != prcsSTATUS_Stopped)
				status = 0;

			if (Process[m->pCfg->HeadCfg.WF.PROC_Indx].Status != prcsSTATUS_Stopped)
				status = 0;

			if (Process[m->pCfg->HeadCfg.GAS.PROC_Indx].Status != prcsSTATUS_Stopped)
				status = 0;

			if (Process[m->pCfg->HeadCfg.WP.PROC_Indx].Status != prcsSTATUS_Stopped)
				status = 0;

			if (Process[m->pCfg->HeadCfg.TIG.PROC_Indx].Status != prcsSTATUS_Stopped)
				status = 0;

			if (Process[m->pCfg->HeadCfg.HW.PROC_Indx].Status != prcsSTATUS_Stopped)
				status = 0;

			if (status)
			{
				LogTxt(&LogMgr, "Prc Final stopped");
				m->SeqStep = 254;
			}

		break;

		case 199: // waiting for signal from OSC

			if (Process[m->pCfg->HeadCfg.OSC.PROC_Indx].fParam[2] == 0.0) // pick is reached
			{

				m->SeqStep = 200;

			}

			if (StopBtn)
			{

				LogTxt(&LogMgr, "Process stop");

				//m->SeqStep = 254;

				//m->SeqStep = 200;

				LogTxt(&LogMgr, "Process stop by Operator");

				Cont_Stop_By_End = 0;

				m->SeqStep = 240;

			}
			else if (ErrorMgr.Error || m->ESTOP)
			{
				LogTxt(&LogMgr, "Process Error");
				m->SeqStep = 100;
			}

		break;

		case 200: // Contin Stop

			// Always Coolant On
			if (!m->TestMode)
			{
				if (Process[m->pCfg->HeadCfg.COOL.PROC_Indx].Status != prcsSTATUS_Run)
					Process[m->pCfg->HeadCfg.COOL.PROC_Indx].xCMD = prcsSTART;
			}

			Process[m->pCfg->HeadCfg.AVC.PROC_Indx].Param[0] = 1; // AVC Locked
			Process[m->pCfg->HeadCfg.TIG.PROC_Indx].Param[1] = 1; // Run Reduce Profile

			Process[m->pCfg->HeadCfg.WF.PROC_Indx].Param[0] = 2; // skip delays & Contin_Ramp
			Process[m->pCfg->HeadCfg.WF.PROC_Indx].xCMD = prcsQuickSTOP;

			Process[m->pCfg->HeadCfg.WP.PROC_Indx].Param[0] = 2; // skip delays & Contin_Ramp
			Process[m->pCfg->HeadCfg.WP.PROC_Indx].xCMD = prcsQuickSTOP;

			Process[m->pCfg->HeadCfg.TVL.PROC_Indx].Param[2] = 4; // Contin_Ramp
			Process[m->pCfg->HeadCfg.TVL.PROC_Indx].xCMD = prcsQuickSTOP;

			Process[m->pCfg->HeadCfg.OSC.PROC_Indx].xCMD = prcsQuickSTOP;

#ifdef EXTENDED_LOGS

			LogTxt(&LogMgr, "Path %d Done: %.2f" , (UDINT)File_RW._int.PathDoneCnt, ABS_TVL_Pos);
#else
			LogTxt(&LogMgr, "Path %d Done" , (UDINT)File_RW._int.PathDoneCnt);

#endif

			//TimerStart(&WF_Catch_TMR, curCfg->Param[parWF_RampDwn].val[0]);
			m->SeqStep++;

		break;

		case 201:

			// Always Coolant On
			if (!m->TestMode)
			{
				if (Process[m->pCfg->HeadCfg.COOL.PROC_Indx].Status != prcsSTATUS_Run)
					Process[m->pCfg->HeadCfg.COOL.PROC_Indx].xCMD = prcsSTART;
			}

			ret = 5; // Preparing To Stop

			if (StopBtn)
			{
#ifdef EXTENDED_LOGS

				LogTxt(&LogMgr, "Quick stop %.2f" , ABS_TVL_Pos);
#else
				LogTxt(&LogMgr, "Quick stop");
#endif
				//m->SeqStep = 254;			// Quick Stop

				LogTxt(&LogMgr, "Process stop by Operator");

				Cont_Stop_By_End = 0;

				m->SeqStep = 240;

				break;

			}

			status = 1;

			if (Process[m->pCfg->HeadCfg.TVL.PROC_Indx].Status != prcsSTATUS_Stopped){ // stopped by end of travel
				status = 0;
			}
			if (Process[m->pCfg->HeadCfg.OSC.PROC_Indx].Status != prcsSTATUS_Stopped){
				status = 0;
			}

			if (Process[m->pCfg->HeadCfg.AVC.PROC_Indx].Status != prcsSTATUS_Stopped){
				//status = 0;
			}

			if (!((Process[m->pCfg->HeadCfg.WF.PROC_Indx].Status == prcsSTATUS_Stopped)
				 || (Process[m->pCfg->HeadCfg.WF.PROC_Indx].Status == prcsSTATUS_Retract))){
				//status = 0;
			}

			if (Process[m->pCfg->HeadCfg.WP.PROC_Indx].Status != prcsSTATUS_Stopped){
				status = 0;
			}

			if (Process[m->pCfg->HeadCfg.TIG.PROC_Indx].Status != prcsSTATUS_Stopped){
				//status = 0;
			}

			if (Process[m->pCfg->HeadCfg.HW.PROC_Indx].Status != prcsSTATUS_Stopped){
				//status = 0;
			}

			if (status)
			{

#ifdef EXTENDED_LOGS

				LogTxt(&LogMgr, "M:All%d Stop: %.2f" ,(UDINT) m->ToolHeadID, ABS_TVL_Pos);

#endif
				switch(curCalib->GenSetup[SETUP_HEAD_SETUP] ){

					/*
					case BPV_v2:
					case BPV_v2_MPBO:
					case BPV_v2_MPGH:
					case BPV_v2_MPGV:

						if(*INDEX_Param_Set[0].pStepDist > 0.0){

							Process[m->pCfg->HeadCfg.OSC.PROC_Indx].xCMD = prcsSTEPpos;

							if(curCalib->GenSetup[SETUP_INDX_DIR])
								Process[m->pCfg->HeadCfg.OSC.PROC_Indx].fParam[1] = (*INDEX_Param_Set[0].pStepDist) * (-1.0);
							else
								Process[m->pCfg->HeadCfg.OSC.PROC_Indx].fParam[1] = (*INDEX_Param_Set[0].pStepDist) ;

							if(m->ToolHeadID == 0){ // Head A make Rewrap so change len of beat B

								if(curCalib->GenDintValue[1]!= 0){

									if(curCalib->GenDintValue[1] < -30)
										curCalib->GenDintValue[1] = -30;

									else if(curCalib->GenDintValue[1] > 30)
										curCalib->GenDintValue[1] = 30;

									Process[m->pCfg->HeadCfg.TVL.PROC_Indx].Param[3] += curCalib->GenDintValue[1]; // Run Length correction

									Process[m->pCfg->HeadCfg.TVL.PROC_Indx].Param[2] = 2; // Rewrap only
									Process[m->pCfg->HeadCfg.TVL.PROC_Indx].xCMD = prcsSTART;

								}

							}else{

								if(curCalib->GenDintValue[0]!= 0){

									if(curCalib->GenDintValue[0] < -30)
										curCalib->GenDintValue[0] = -30;

									else if(curCalib->GenDintValue[0] > 30)
										curCalib->GenDintValue[0] = 30;

									Process[m->pCfg->HeadCfg.TVL.PROC_Indx].Param[3] += curCalib->GenDintValue[0]; // Run Length correction

									Process[m->pCfg->HeadCfg.TVL.PROC_Indx].Param[2] = 2; // Rewrap only
									Process[m->pCfg->HeadCfg.TVL.PROC_Indx].xCMD = prcsSTART;

								}
							}

							KK_Catched = 133;

						}

					break;
					*/

					default:

						if(curCalib->GenSetup[SETUP_INDX_ENBL] == 3){ // In OSc

							/*
							if(INDEX_Param_Set[0].pStepDist){

								Process[m->pCfg->HeadCfg.OSC.PROC_Indx].xCMD = prcsSTEPpos;

								if(curCalib->GenSetup[SETUP_INDX_DIR])
									Process[m->pCfg->HeadCfg.OSC.PROC_Indx].fParam[1] = (*INDEX_Param_Set[0].pStepDist);
								else
									Process[m->pCfg->HeadCfg.OSC.PROC_Indx].fParam[1] = (*INDEX_Param_Set[0].pStepDist) * (-1.0);

								KK_Catched = 133;

								m->SeqStep++;
							}
							else
								m->SeqStep = 203;

							*/

								if(*INDEX_Param_Set[0].pStepDist > 0.0){

								Process[m->pCfg->HeadCfg.OSC.PROC_Indx].xCMD = prcsSTEPpos;

								if(curCalib->GenSetup[SETUP_INDX_DIR])
									Process[m->pCfg->HeadCfg.OSC.PROC_Indx].fParam[1] = (*INDEX_Param_Set[0].pStepDist) * (-1.0);
								else
									Process[m->pCfg->HeadCfg.OSC.PROC_Indx].fParam[1] = (*INDEX_Param_Set[0].pStepDist) ;

								if(m->ToolHeadID == 0){ // Head A make Rewrap so change len of beat B

									if(curCalib->GenDintValue[1]!= 0){

										if(curCalib->GenDintValue[1] < -30)
											curCalib->GenDintValue[1] = -30;

										else if(curCalib->GenDintValue[1] > 30)
											curCalib->GenDintValue[1] = 30;

										Process[m->pCfg->HeadCfg.TVL.PROC_Indx].Param[3] += curCalib->GenDintValue[1]; // Run Length correction

										Process[m->pCfg->HeadCfg.TVL.PROC_Indx].Param[2] = 2; // Rewrap only
										Process[m->pCfg->HeadCfg.TVL.PROC_Indx].xCMD = prcsSTART;

									}

								}else{

									if(curCalib->GenDintValue[0]!= 0){

										if(curCalib->GenDintValue[0] < -30)
											curCalib->GenDintValue[0] = -30;

										else if(curCalib->GenDintValue[0] > 30)
											curCalib->GenDintValue[0] = 30;

										Process[m->pCfg->HeadCfg.TVL.PROC_Indx].Param[3] += curCalib->GenDintValue[0]; // Run Length correction

										Process[m->pCfg->HeadCfg.TVL.PROC_Indx].Param[2] = 2; // Rewrap only
										Process[m->pCfg->HeadCfg.TVL.PROC_Indx].xCMD = prcsSTART;

									}
								}

								KK_Catched = 133;

							}

						}

						else if(curCalib->GenSetup[SETUP_INDX_ENBL] == 1){

							if(INDEX_Param_Set[0].pStepDist){
								Process[m->pCfg->HeadCfg.INDX.PROC_Indx].xCMD = prcsSTEPpos;

								if(curCalib->GenSetup[SETUP_INDX_DIR])
									Process[m->pCfg->HeadCfg.INDX.PROC_Indx].fParam[1] = (*INDEX_Param_Set[0].pStepDist);
								else
									Process[m->pCfg->HeadCfg.INDX.PROC_Indx].fParam[1] = (*INDEX_Param_Set[0].pStepDist) * (-1.0);

								m->SeqStep++;

							}
							else
								m->SeqStep = 203;

						}
						else
							m->SeqStep = 203;

					break;

				}

				//m->SeqStep = 203;
				m->SeqStep = 230;

			}

		break;

		/////////////////////////////////////////////////////////////////////////////////////
		/////////////////////////////////////////////////////////////////////////////////////
		case 230: // Start New Path

			if (StopBtn)
			{
				LogTxt(&LogMgr, "Quick stop");

				//m->SeqStep = 254;			// Quick Stop

				LogTxt(&LogMgr, "Process stop by Operator");

				Cont_Stop_By_End = 0;

				m->SeqStep = 240;

				break;
			}

			if(Process[m->pCfg->HeadCfg.OSC.PROC_Indx].Status != prcsSTATUS_Stopped)
				break;

			if(Process[m->pCfg->HeadCfg.TVL.PROC_Indx].Status != prcsSTATUS_Stopped)
				break;

			// New Path in New Direction

			m->ToolHeadID = !m->ToolHeadID;

			CalculateRunOverlap_Cont();

			Process[m->pCfg->HeadCfg.TVL.PROC_Indx].Param[2] = 4; // Contin_Ramps
			Process[m->pCfg->HeadCfg.TVL.PROC_Indx].xCMD = prcsQuickStart;

			Process[m->pCfg->HeadCfg.OSC.PROC_Indx].xCMD = prcsJump2Run;

			Process[m->pCfg->HeadCfg.TIG.PROC_Indx].Param[1] = 0; // return from Reduce Profile

			Process[m->pCfg->HeadCfg.AVC.PROC_Indx].Param[0] = 0; // AVC UnLocked

			if (!m->WireDisabled){
				Process[m->pCfg->HeadCfg.WF.PROC_Indx].xCMD = prcsQuickStart;
				Process[m->pCfg->HeadCfg.WF.PROC_Indx].Param[0] = 2; // skip delays & Contin Ramps
				Process[m->pCfg->HeadCfg.WP.PROC_Indx].xCMD = prcsQuickStart;
				Process[m->pCfg->HeadCfg.WP.PROC_Indx].Param[0] = 2; // skip delays & Contin Ramps
			}

#ifdef EXTENDED_LOGS
			LogTxt(&LogMgr, "M:TVL%d Start: %.2f" , (UDINT) m->ToolHeadID , ABS_TVL_Pos);
#endif
			StartPos = 0;

			m->SeqStep = 3;

		break;

		///////////////   Stop By Operator
		//////////////////////////////////////////////////////////////////////////////
		case 240: // Stop by Btn

			// Always Coolant On
			if (!m->TestMode)
			{
				if (Process[m->pCfg->HeadCfg.COOL.PROC_Indx].Status != prcsSTATUS_Run)
					Process[m->pCfg->HeadCfg.COOL.PROC_Indx].xCMD = prcsSTART;
			}

			for (i = 0; i < PROCESS_NUM; i++)
			{
				if ((i != PROC_COOL)) //&&( i != m->pCfg->HeadCfg.TVL.PROC_Indx))
					Process[i].xCMD = prcsSTOP;

			}

			Process[m->pCfg->HeadCfg.TVL.PROC_Indx].Param[2] = 0; // Regular stop no retract a moze byc z 1 wtedy rewrap
			Process[m->pCfg->HeadCfg.WF.PROC_Indx].Param[0] = 1; // Regular stop no retract
			Process[m->pCfg->HeadCfg.WP.PROC_Indx].Param[0] = 1; // Regular stop no retract

#ifdef EXTENDED_LOGS

			LogTxt(&LogMgr, "Path %d Done: %.2f" , (UDINT)File_RW._int.PathDoneCnt, ABS_TVL_Pos);
#else
			LogTxt(&LogMgr, "Path %d Done" , (UDINT)File_RW._int.PathDoneCnt);

#endif

			//TimerStart(&WF_Catch_TMR, curCfg->Param[parWF_RampDwn].val[0]);
			m->SeqStep++;

		break;

		case 241:

			// Always Coolant On
			if (!m->TestMode)
			{
				if (Process[m->pCfg->HeadCfg.COOL.PROC_Indx].Status != prcsSTATUS_Run)
					Process[m->pCfg->HeadCfg.COOL.PROC_Indx].xCMD = prcsSTART;
			}

			ret = 5; // Preparing To Stop

			if (StopBtn)
			{
#ifdef EXTENDED_LOGS

				LogTxt(&LogMgr, "Quick stop %.2f" , ABS_TVL_Pos);
#else
				LogTxt(&LogMgr, "Quick stop");
#endif
				m->SeqStep = 254;			// Quick Stop
			}

			status = 1;

			if (Process[m->pCfg->HeadCfg.TVL.PROC_Indx].Status != prcsSTATUS_Stopped){ // stopped by end of travel
				status = 0;
			}
			if (Process[m->pCfg->HeadCfg.OSC.PROC_Indx].Status != prcsSTATUS_Stopped)
				status = 0;

			if (Process[m->pCfg->HeadCfg.AVC.PROC_Indx].Status != prcsSTATUS_Stopped)
				status = 0;

			if (Process[m->pCfg->HeadCfg.WF.PROC_Indx].Status != prcsSTATUS_Stopped)
				status = 0;

			//if (Process[m->pCfg->HeadCfg.GAS.PROC_Indx].Status != prcsSTATUS_Stopped)
				//status = 0;

			if (Process[m->pCfg->HeadCfg.WP.PROC_Indx].Status != prcsSTATUS_Stopped)
				status = 0;

			if (Process[m->pCfg->HeadCfg.TIG.PROC_Indx].Status != prcsSTATUS_Stopped)
				status = 0;

			if (Process[m->pCfg->HeadCfg.HW.PROC_Indx].Status != prcsSTATUS_Stopped)
				status = 0;

			if (status)
			{

#ifdef EXTENDED_LOGS

				LogTxt(&LogMgr, "M:All%d Stop: %.2f" ,(UDINT) m->ToolHeadID, ABS_TVL_Pos);

#endif
				m->SeqStep++;

			}

		break;

		case 242:

			// Always Coolant On
			if (!m->TestMode)
			{
				if (Process[m->pCfg->HeadCfg.COOL.PROC_Indx].Status != prcsSTATUS_Run)
					Process[m->pCfg->HeadCfg.COOL.PROC_Indx].xCMD = prcsSTART;
			}

			if (StopBtn)
			{
				LogTxt(&LogMgr, "Quick stop");

				m->SeqStep			= 254;			// Quick Stop
				break;
			}

			if(Process[m->pCfg->HeadCfg.INDX.PROC_Indx].Status == prcsSTATUS_Stopped
				&& Process[m->pCfg->HeadCfg.OSC.PROC_Indx].Status == prcsSTATUS_Stopped){

				TimerStart(&m->sm.Tmr1, 0.1);
				m->SeqStep++;

			}

		break;

		case 243:
			// Always Coolant On
			if (StopBtn)
			{
				LogTxt(&LogMgr, "Halt stop");

				m->SeqStep			= 254;			// Quick Stop
				break;
			}

			if (!m->TestMode)
			{
				if (Process[m->pCfg->HeadCfg.COOL.PROC_Indx].Status != prcsSTATUS_Run)
					Process[m->pCfg->HeadCfg.COOL.PROC_Indx].xCMD = prcsSTART;
			}

			if(Process[m->pCfg->HeadCfg.TVL.PROC_Indx].Status == prcsSTATUS_Stopped){

				LogTxt(&LogMgr, "M: Cyc. Time %.2f" , GlobalTimer);

				if(Cont_Stop_By_End)
					m->ToolHeadID = !m->ToolHeadID;

				if(Cont_Stop_By_End){
					m->SeqStep++;
				}
				else{

					m->SeqStep = 0;
				}

			}

		break;

		/////////////////////////////////////////////////////////////////////////////////////////////////////

		case 244:

			switch(curCalib->GenSetup[SETUP_HEAD_SETUP] ){

					/*
					case BPV_v2_MPGH:
					case BPV_v2_MPGV:

					case BPV_v2_MPBO:
					*/

					default:

						if(*INDEX_Param_Set[0].pStepDist > 0.0){

							Process[m->pCfg->HeadCfg.OSC.PROC_Indx].xCMD = prcsSTEPpos;

							if(curCalib->GenSetup[SETUP_INDX_DIR])
								Process[m->pCfg->HeadCfg.OSC.PROC_Indx].fParam[1] = (*INDEX_Param_Set[0].pStepDist) * (-1.0);
							else
								Process[m->pCfg->HeadCfg.OSC.PROC_Indx].fParam[1] = (*INDEX_Param_Set[0].pStepDist) ;

							KK_Catched = 135;

						}

					break;

				}

				m->SeqStep = 0;

		break;

		/////////////////////////////////////////////////////////////////////////////

		case 254: // Quick End of Welding

			for (i = 0; i < PROCESS_NUM; i++)
			{ // beside PROC_COOL
				if (i != PROC_COOL)
					Process[i].xCMD = prcsHalt;
			}

			Process[m->pCfg->HeadCfg.OSC.PROC_Indx].Param[0] = 1; // STop without ramp
			Process[m->pCfg->HeadCfg.OSC.PROC_Indx].xCMD = prcsQuickSTOP; // return to center position
			Process[m->pCfg->HeadCfg.GAS.PROC_Indx].xCMD = prcsSTOP; // maintain gas
			m->SeqStep++;

		break;

		default:

			if(curCfg->Param_ENUM[parENUM_AVC_Mode].val[0] != 3) // AVC Mode NOT LOCKED !
				Process[m->pCfg->HeadCfg.AVC.PROC_Indx].Param[0] = 0;

			if (StopBtn)
			{
				LogTxt(&LogMgr, "Halt stop");

				for (i = 0; i < PROCESS_NUM; i++)
				{ // beside PROC_COOL
					if (i!= PROC_COOL && i!= PROC_OSC)
						Process[i].xCMD = prcsHalt;
				}

				Process[m->pCfg->HeadCfg.GAS.PROC_Indx].xCMD = prcsSTOP; // maintain gas
				m->SeqStep			= 0;

			}

			if (Process[m->pCfg->HeadCfg.OSC.PROC_Indx].Status == prcsSTATUS_Stopped)
				m->SeqStep = 0;

			if (m->SeqStep == 0)
			{
				// Load new AVC param from new file
				TML_MTR_INST[m->pCfg->HeadCfg.AVC.TML_A_Indx]._cfg.signFilter =	curCfg->Param[parAVC_FbkFilter].val[0];
			}

		break;

		}

		//if((Process[m->pCfg->HeadCfg.TVL.PROC_Indx].Status == prcsSTATUS_Stopped))
		//StopBtn_Latch = 0;
		////////////////////////////
		TimerExecute(&WireDisable_TMR);
		TimerExecute(&WF_Catch_TMR);

		return ret;
	}

void ProcessEvents_Android(MASTER_typ * m, LCD_NODE_obj * nodes, HMI_typ * hmi, HMI_INTRF_typ * intrf)
{
USINT			status;
UINT			where, indx, seg;
Scaled_Var_obj * pVar;
int 			i, k;
float			x, y, z, a, A, b, B;
CurCfg_typ *	curCfg;

UINT segm;
float pos;

//float TVL_StopDly , TVL_RmpDwn ,TVL_Vel , TVL_Vel_Fin , TVL_ReWrap;
//float WF_StopDly , WF_RmpDwn;
curCfg				= m->pCurCfg;

	if (!curCfg)
		return;

	if (File_RW.NewFileLoaded)
	{

		File_RW.NewFileLoaded = 0;

		hmi->PLC_Changes	|= (0x0001 + 0x0002 + 0x0004 + 0x0008); // New CurCfg and New segment List

		PleaseUpdateHeadSetup(m);

		_TIG_Mode = 0xFFFF;
		_AVC_Mode = 0xFFFF;

		// Force limits from Cfg in curCfg for enumerated values
		for (i = 0; i < m->paramEnumLastNum; i++)
		{
			curCfg->Param_ENUM[i].min = cfg->Param_ENUM[i].min;
			curCfg->Param_ENUM[i].max = cfg->Param_ENUM[i].max;

		}

	}

	switch (hmi->FiredEvent)
	{

			case EVNT_SET_INDX_ZERO:

			switch(curCalib->GenSetup[SETUP_HEAD_SETUP]){

				case BPV_F_HEAD:
				case CLAMSHELL_HEAD:
				case CHERRYPOINT_BP1_HEAD:
				case CHERRYPOINT_BP2_HEAD:
				case CHERRYPOINT_MT_BP2_HEAD:
				case MIG_TIG_HEAD:
				//dodane 6Dec23
				case BPV_v1_MT:

					VectorStateMach[m->pCfg->HeadCfg.INDX.VECT_A_Indx].Param[0] = 0;
					VectorStateMach[m->pCfg->HeadCfg.INDX.VECT_A_Indx].xCMD = VECT_Set_Act_Pos;

					VectorStateMach[m->pCfg->HeadCfg.INDX.VECT_B_Indx].Param[0] = 0;
					VectorStateMach[m->pCfg->HeadCfg.INDX.VECT_B_Indx].xCMD = VECT_Set_Act_Pos;

					strcpy(hmi->pMessage[0], "	INDEX ");
					strcpy(hmi->pMessage[1], "	Zero ");
					xsprintf(hmi->pMessage[2], "is Set");
					strcpy(hmi->pMessage[3], " ");
					TimerStart(&hmi->MsgTmr, 0.1);

				break;

				case BPV_v2:
				case BPV_v2_Video:
				case BPV_v2_MPBO:
				case BPV_v2_MPGH:
				case BPV_v2_MPGV:
				//dodane 6Dec23
				case BPV_v2_MT:

					TML_MTR_INST[m->pCfg->HeadCfg.INDX.TML_A_Indx]._cfg.absLastPos = 0; //OLD_MTR_POS[INDX_B_LAST_POS];
					TML_MTR_INST[m->pCfg->HeadCfg.INDX.TML_A_Indx]._cfg.absFbk = 2;
					TML_MTR_INST[m->pCfg->HeadCfg.INDX.TML_A_Indx].xCMD = 1;

					TML_MTR_INST[m->pCfg->HeadCfg.INDX.TML_B_Indx]._cfg.absLastPos = 0; //OLD_MTR_POS[INDX_B_LAST_POS];
					TML_MTR_INST[m->pCfg->HeadCfg.INDX.TML_B_Indx]._cfg.absFbk = 2;
					TML_MTR_INST[m->pCfg->HeadCfg.INDX.TML_B_Indx].xCMD = 1;

					strcpy(hmi->pMessage[0], "	INDEX ");
					strcpy(hmi->pMessage[1], "	Zero ");
					xsprintf(hmi->pMessage[2], "is Set");
					strcpy(hmi->pMessage[3], " ");
					TimerStart(&hmi->MsgTmr, 0.1);

				break;

				default:

					strcpy(hmi->pMessage[0], "	INDEX ");
					strcpy(hmi->pMessage[1], "	is Not");
					xsprintf(hmi->pMessage[2], "Allowed");
					strcpy(hmi->pMessage[3], " in this head ");
					TimerStart(&hmi->MsgTmr, 0.1);

				break;

			}

			break;

			//////////////////////////////////////////////////////////////////
			case EVNT_FILL_MODE:

				curCalib->GenSetup[SETUP_OSC_EXC_MODE] ++;

				if (curCalib->GenSetup[SETUP_OSC_EXC_MODE] > 2)
					curCalib->GenSetup[SETUP_OSC_EXC_MODE] = 0;

			break;

			////////////////////////////////////////////////////////////////////
			case EVENT_WELD_WIZARD_DONE:

				strcpy(hmi->pMessage[0], "	  WIZARD");
				strcpy(hmi->pMessage[1], "	Calculated ");
				xsprintf(hmi->pMessage[2], "New Timing");
				strcpy(hmi->pMessage[3], " ");
				TimerStart(&hmi->MsgTmr, 0.1);

			break;

			////////////////////////////////////////////////////////////////////
			case EVNT_STEP_FWD:

				if (Process[m->pCfg->HeadCfg.TVL.PROC_Indx].Status == prcsSTATUS_Stopped)
					Process[m->pCfg->HeadCfg.TVL.PROC_Indx].xCMD = prcsSTEPpos;

			break;

			////////////////////////////////////////////////////////////////////
			case EVNT_STEP_REV:

				if (Process[m->pCfg->HeadCfg.TVL.PROC_Indx].Status == prcsSTATUS_Stopped)
					Process[m->pCfg->HeadCfg.TVL.PROC_Indx].xCMD = prcsSTEPneg;

			break;

			////////////////////////////////////////////////////////////////////
			case EVNT_TEST_MODE_ON_OFF:

				if (m->SeqStep == 0)
				{
					if (intrf->TestMode != 0)
						intrf->TestMode = 0;
					else
						intrf->TestMode = 1;
				}

			break;

			////////////////////////////////////////////////////////////////////
			case EVNT_SWAP_HEAD:

				if (m->SeqStep != 0) // No Head Changes on run
					break;

				if (m->ToolHeadID != 0)
					m->ToolHeadID = 0;
				else
					m->ToolHeadID = 1;

				if(curCalib->GenSetup[SETUP_TVL_ENC_SET]){
					if (TVL_ROT_Param_Set[0].pEncoder)
						OLD_MTR_POS[TVL_ENC_HOME] = *TVL_ROT_Param_Set[0].pEncoder;
				}

				m->SubSeqStep = 1;

			break;

			////////////////////////////////////////////////////////////////////
			case EVNT_SAVE_CURCFG:

				if (File_RW.CMD == 0)
				{
					File_RW.CMD = F_SAVE_CURCFG;

					strcpy(hmi->pMessage[0], "	  Parameters  ");
					strcpy(hmi->pMessage[1], "	 ");
					strcpy(hmi->pMessage[2], "		SAVED ");
					strcpy(hmi->pMessage[3], " ");
					TimerStart(&hmi->MsgTmr, 1.0);

				}

			break;

			////////////////////////////////////////////////////////////////////

			case EVNT_POPUP_OK:

				switch(POPUP_EVENT){

					case EVNT_SET_HOME:

						SetZeroPosition(m);

						strcpy(hmi->pMessage[0], "Segm and TVL Zero ");
						strcpy(hmi->pMessage[1], " are Set ");
						xsprintf(hmi->pMessage[2], "");
						strcpy(hmi->pMessage[3], "");
						TimerStart(&hmi->MsgTmr, 0.5);
						//KK_test = 2;

					break;

					case EVNT_OSC_ALLIGMENT:

						if(OSC_TML_Param_Set[0].PosFbkIndx == 2)
							pos = OSC_TML_Param_Set[0].pVect->FbkVect.x2 ;

						else
							pos = OSC_TML_Param_Set[0].pVect->FbkVect.x ;

						if((*OSC_TML_Param_Set[0].pPrimAmpl) > (OSC_TML_Param_Set[0].pVect->OutVect.softLimits[1] - OSC_TML_Param_Set[0].pVect->OutVect.softLimits[0]))
							(*OSC_TML_Param_Set[0].pPrimAmpl) = (OSC_TML_Param_Set[0].pVect->OutVect.softLimits[1] - OSC_TML_Param_Set[0].pVect->OutVect.softLimits[0]);

						if((pos  + (*OSC_TML_Param_Set[0].pPrimAmpl)/2.0) > OSC_TML_Param_Set[0].pVect->OutVect.softLimits[1]){

							(*OSC_TML_Param_Set[0].pPrimAmpl) = (OSC_TML_Param_Set[0].pVect->OutVect.softLimits[1] - pos )*2.0;
						}

						else if((pos  - (*OSC_TML_Param_Set[0].pPrimAmpl)/2) < OSC_TML_Param_Set[0].pVect->OutVect.softLimits[0]){

							(*OSC_TML_Param_Set[0].pPrimAmpl) = (pos  - OSC_TML_Param_Set[0].pVect->OutVect.softLimits[0])*2.0;

						}

						// Check if Amplitude not negative
						if((*OSC_TML_Param_Set[0].pPrimAmpl) < 0)
							(*OSC_TML_Param_Set[0].pPrimAmpl) = 0;

					break;

				}

				POPUP_EVENT = 0;

			break;

			case EVNT_POPUP_CANCEL:

				switch(POPUP_EVENT){

					case EVNT_SET_HOME:

						//KK_test = 3;

					break;

					case EVNT_OSC_ALLIGMENT:

						Process[m->pCfg->HeadCfg.OSC.PROC_Indx].xCMD = prcsAlligment;

					break;

				}
				POPUP_EVENT = 0;

			break;

			case EVNT_SET_HOME:

				if (m->SeqStep == 0)
				{
					POPUP_EVENT = EVNT_SET_HOME;

					if (TVL_ROT_Param_Set[0].pEncoder)
						OLD_MTR_POS[TVL_ENC_HOME] = *TVL_ROT_Param_Set[0].pEncoder;

					VectorStateMach[m->pCfg->HeadCfg.INDX.VECT_A_Indx].Param[0] = 0;
					VectorStateMach[m->pCfg->HeadCfg.INDX.VECT_A_Indx].xCMD = VECT_Set_Act_Pos;

					VectorStateMach[m->pCfg->HeadCfg.INDX.VECT_B_Indx].Param[0] = 0;
					VectorStateMach[m->pCfg->HeadCfg.INDX.VECT_B_Indx].xCMD = VECT_Set_Act_Pos;

					strcpy(hmi->pMessage[0], "TVL Zero is Set. ");
					strcpy(hmi->pMessage[1], "Do you want to Set ");
					xsprintf(hmi->pMessage[2], "Segment Zero");
					strcpy(hmi->pMessage[3], " as well ?");
					hmi->xCMD = SHOW_POPUP_CMD;

				}else{

					strcpy(hmi->pMessage[0], "  Sorry,");
					strcpy(hmi->pMessage[1], " I am not");
					xsprintf(hmi->pMessage[2], "  ready");
					strcpy(hmi->pMessage[3], "");
					TimerStart(&hmi->MsgTmr, 0.5);

				}

			break;

			////////////////////////////////////////////////////////////////////
			case EVNT_TEST_OSC:

				if (m->SeqStep == 0)
				{

					if (Process[m->pCfg->HeadCfg.OSC.PROC_Indx].Status == prcsSTATUS_Stopped)
					{
						if(Check_OSC_Amplt_and_Center()){

							Process[m->pCfg->HeadCfg.OSC.PROC_Indx].Param[0] = 1; // Start without ramp
							Process[m->pCfg->HeadCfg.OSC.PROC_Indx].xCMD = prcsJump2Run;

						}
					}
					else if (Process[m->pCfg->HeadCfg.OSC.PROC_Indx].Status == prcsSTATUS_Run)
					{
						Process[m->pCfg->HeadCfg.OSC.PROC_Indx].Param[0] = 1; // Stop without ramp
						Process[m->pCfg->HeadCfg.OSC.PROC_Indx].xCMD = prcsQuickSTOP;

					}

				}

			break;

			////////////////////////////////////////////////////////////////////
			case EVNT_GAS_ON_OFF:

				if (m->Mode != MASTER_MODE_RUN)
				{
					if (Process[m->pCfg->HeadCfg.GAS.PROC_Indx].Status == prcsSTATUS_Stopped)
						Process[m->pCfg->HeadCfg.GAS.PROC_Indx].xCMD = prcsForceON;

					else if (Process[m->pCfg->HeadCfg.GAS.PROC_Indx].Status == prcsSTATUS_Run)
						Process[m->pCfg->HeadCfg.GAS.PROC_Indx].xCMD = prcsHalt;
				}

			break;

			////////////////////////////////////////////////////////////////////
			case EVNT_GO_CALIB_MODE:

				if((Process[m->pCfg->HeadCfg.GAS.PROC_Indx].Status != prcsSTATUS_Stopped) ||
					(Process[m->pCfg->HeadCfg.AVC.PROC_Indx].Status != prcsSTATUS_Stopped) ||
					(Process[m->pCfg->HeadCfg.OSC.PROC_Indx].Status != prcsSTATUS_Stopped) ||
					(Process[m->pCfg->HeadCfg.TVL.PROC_Indx].Status != prcsSTATUS_Stopped) ||
					(Process[m->pCfg->HeadCfg.WF.PROC_Indx].Status != prcsSTATUS_Stopped) ||
					(Process[m->pCfg->HeadCfg.WP.PROC_Indx].Status != prcsSTATUS_Stopped))
					status = 0;

				if (status && (m->sm.Step == 50))
				{
					m->sm.Step = 100;
				}

			break;

			////////////////////////////////////////////////////////////////////
		case EVNT_RETURN_CALIB_MODE:

			for (i = 0; i < PROCESS_NUM; i++)
			{ // beside PROC_COOL
				if (i != PROC_COOL)
					Process[i].xCMD = prcsHalt;
			}

			Process[m->pCfg->HeadCfg.GAS.PROC_Indx].xCMD = prcsSTOP; // rmaintain gas
			m->sm.Step = 0;

		break;

		/////////////////////////////////////////////////////////////////////////////////
		case EVNT_OSC_POS_LIMIT_SET:

			if (m->pCfg->HeadCfg.OSC.Limits_Harcoded)
			{

				strcpy(hmi->pMessage[0], " OSC Limits  ");
				strcpy(hmi->pMessage[1], " are hardcoded  ");
				strcpy(hmi->pMessage[2], " Operation ");
				strcpy(hmi->pMessage[3], " denied");
				TimerStart(&hmi->MsgTmr, 1.5);

				break;

			}

			if((curCalib->GenSetup[SETUP_HEAD_SETUP] == BPV_v2_MT_BO_TOS)
				|| (curCalib->GenSetup[SETUP_HEAD_SETUP] == BPV_v2_TT_BO_TOS)
				|| (curCalib->GenSetup[SETUP_HEAD_SETUP] == BPV_v2_MPGH)
				|| (curCalib->GenSetup[SETUP_HEAD_SETUP] == BPV_v2_MPGV) ){

					curCalib->Points[CALIB_OSC_SFT_LIMIT].val[1] = TML_MTR_INST[m->pCfg->HeadCfg.TVL.TML_Indx].PosFBK;

					strcpy(hmi->pMessage[0], " TVL (OSC) Positive  ");
					strcpy(hmi->pMessage[1], " Software  ");
					strcpy(hmi->pMessage[2], " Limit SET ");
					strcpy(hmi->pMessage[3], " ");
					TimerStart(&hmi->MsgTmr, 1.5);
```
